PROGRAM F01_METS_SingleInputs
VAR
(*METS General Filtered Inputs FB ***************************************************************************************************************)

	fbMestStart				: 	FB_IO2_SingleInputCtrl;
	fbMestStop				: 	FB_IO2_SingleInputCtrl;
	fbMestReset				:	FB_IO2_SingleInputCtrl;

	fbMETS_24VPowerSupplyOK		: FB_IO2_SingleInputCtrl;
	fbTPD24VPowerSupplyOK			: FB_IO2_SingleInputCtrl;
	fbAirPressureOK				: FB_IO2_SingleInputCtrl;
	fbAirConditionerOK				: FB_IO2_SingleInputCtrl; (**)
	fbUPSBatteryAlarm				: FB_IO2_SingleInputCtrl;
	fbNetworkOKFromSwitch			: FB_IO2_SingleInputCtrl;


	fbPreMachineAutoRun			: FB_IO2_SingleInputCtrl;
	fbCasePackerAutoRun			: FB_IO2_SingleInputCtrl;

	fbDoorOpenZone1				: FB_IO2_SingleInputCtrl;
	fbDoorOpenZone2 				: FB_IO2_SingleInputCtrl;

	fbAuxRowCompleteSesnor			: FB_IO2_SingleInputCtrl;
	fbCaseAtRejectStation	 		: FB_IO2_SingleInputCtrl;
	fbCaseRejectedByCasePacker		: FB_IO2_SingleInputCtrl;
	fbCaseContentValidationComplete	: FB_IO2_SingleInputCtrl;
	fbCaseLeavingPrintArea			: FB_IO2_SingleInputCtrl;

(*METS CX UPS  Filtered Inputs  FB***************************************************************************************************************)
	fbMainSupplyHealthy			:	FB_IO2_SingleInputCtrl;	(*ib64KF1_1_MainsSupplyHealthy*)
	fbUPSHealthy					:	FB_IO2_SingleInputCtrl;	(*ib64KF1_5_UPSHealthy*)
	fbUPSBatteryMode				:	FB_IO2_SingleInputCtrl;	(*ib64KF1_2_UPSBatteryMode*)
	fbUPSBatteryCharging			:	FB_IO2_SingleInputCtrl;	(*ib64KF1_6_UPSBatteryCharging*)


(*METS Camera Filtered Inputs  FB***************************************************************************************************************)

	fbCamera01TrigSensor			: FB_IO2_SingleInputCtrl;
	fbCamera02TrigSensor			: FB_IO2_SingleInputCtrl;
	fbCamera03TrigSensor			: FB_IO2_SingleInputCtrl;
	fbCamera04TrigSensor			: FB_IO2_SingleInputCtrl;
	fbCamera05TrigSensor			: FB_IO2_SingleInputCtrl;
	fbCamera06TrigSensor			: FB_IO2_SingleInputCtrl;
	fbCamera07TrigSensor			: FB_IO2_SingleInputCtrl;
	fbCamera08TrigSensor			: FB_IO2_SingleInputCtrl;
	fbCamera09TrigSensor			: FB_IO2_SingleInputCtrl;
	fbCamera10TrigSensor			: FB_IO2_SingleInputCtrl;
	fbCamera11TrigSensor			: FB_IO2_SingleInputCtrl;
	fbCamera12TrigSensor			: FB_IO2_SingleInputCtrl;

(*METS Casepacker  Filtered Inputs  FB***************************************************************************************************************)

	fbEUCABuildBackPreMachine		: FB_IO2_SingleInputCtrl;
	fbEUCAExitBlocked				: FB_IO2_SingleInputCtrl; (**)

	fbOuterAtSystemInfeed		: FB_IO2_SingleInputCtrl;
	fbOuterAtAdditionalConv		: FB_IO2_SingleInputCtrl;

	fbQAButtonReject				: FB_IO2_SingleInputCtrl;
	fbOuterAtRejectStation 			: FB_IO2_SingleInputCtrl;
	fbOuterRejectConfirm			: FB_IO2_SingleInputCtrl;
	fbRejectBinFull					: FB_IO2_SingleInputCtrl;


	(*Transfer Conveyor*)
	fbTransferCoveyorDoorGuard1		: FB_IO2_SingleInputCtrl;
	fbTransferCoveyorDoorGuard2		: FB_IO2_SingleInputCtrl;

	fbTransferConveyorPlugConnected	: FB_IO2_SingleInputCtrl;
	fbOutfeedConveyorPlugConnected	: FB_IO2_SingleInputCtrl;
	fbAdditionalConveyorPlugConnected	: FB_IO2_SingleInputCtrl;



(*METS Cylinders Filtered Inputs  FB***************************************************************************************************************)

	fbClampCylinderExtended		: FB_IO2_SingleInputCtrl;
	fbClampCylinderRetracted		: FB_IO2_SingleInputCtrl;

	fbGateCylinderExtended			: FB_IO2_SingleInputCtrl;
	fbGateCylinderRetracted 			: FB_IO2_SingleInputCtrl;

	fbRejectCylinderExtended		: FB_IO2_SingleInputCtrl;
	fbRejectCylinderRetracted 		: FB_IO2_SingleInputCtrl;

	fbAdditionalRejectCylinderExtended		: FB_IO2_SingleInputCtrl;
	fbAdditionalRejectCylinderRetracted 		: FB_IO2_SingleInputCtrl;

	fbFirstPusherCylinderExtended		: FB_IO2_SingleInputCtrl;
	fbFirstPusherCylinderRetracted 		: FB_IO2_SingleInputCtrl;

	fbSecondPusherCylinderExtended		: FB_IO2_SingleInputCtrl;
	fbSecondPusherCylinderRetracted 		: FB_IO2_SingleInputCtrl;

(*METS SFLX Machine Filtered Inputs  FB***************************************************************************************************************)

	fbOuterInfeedJam						: FB_IO2_SingleInputCtrl;
	fbOuterTransferConfirmation			: FB_IO2_SingleInputCtrl;
	fbRejectConfirmationNCW				: FB_IO2_SingleInputCtrl;
	fbRejectBinFullNCW					: FB_IO2_SingleInputCtrl;
	fbOuterAtTransferReject				: FB_IO2_SingleInputCtrl;
	fbOuterAtSideFlexExit					: FB_IO2_SingleInputCtrl;
	fbOuterAtPostMachineInfeed			: FB_IO2_SingleInputCtrl;

	fbGuard1FlexInfeedDoor	  	: FB_IO2_SingleInputCtrl;
	fbGuard3FlexRHDoor		: FB_IO2_SingleInputCtrl;
	fbGuard4FlexPrinterDoor		: FB_IO2_SingleInputCtrl;
	fbGuard5FlexLHDoor		: FB_IO2_SingleInputCtrl;

(*METS CML Filtered Inputs ***************************************************************************************************************)

	fbGuard1UpperSideAccessDoor	: FB_IO2_SingleInputCtrl;
	fbGuard2UpperDoorLabellerSide	: FB_IO2_SingleInputCtrl;
	fbGuard3OutfeedTunnel			: FB_IO2_SingleInputCtrl;
	fbGuard4ElectricalBoxInPosition	: FB_IO2_SingleInputCtrl;
	fbGuard5RejectBinLHSide			: FB_IO2_SingleInputCtrl;
	fbGuard6RejectBinRHSide			: FB_IO2_SingleInputCtrl;
	fbGuard7HTTDoorGuard			: FB_IO2_SingleInputCtrl;
	fbGuard10FrontUpperDoor			: FB_IO2_SingleInputCtrl;
	fbGuard11GuardLowerLabellerSide	: FB_IO2_SingleInputCtrl;

	fbRejectBinGuardIsReset			: FB_IO2_SingleInputCtrl;
	fbLabeller1GuardIsReset			: FB_IO2_SingleInputCtrl;
	fbLabeller2GuardIsReset			: FB_IO2_SingleInputCtrl;

	fbResetPB							: FB_IO2_SingleInputCtrl;

	fbOuterAtCMLRejectStation		: FB_IO2_SingleInputLockCtrl;

	fbRotaryTransferPackAtStopPlate		: FB_IO2_SingleInputCtrl;
	fbRotaryTransferTorqueLimiter		: FB_IO2_SingleInputCtrl;
	fbRotaryTransferDelayStop1			: FB_IO2_SingleInputCtrl;
	fbRotaryTransferDelayStop2			: FB_IO2_SingleInputCtrl;

	fbLoweratorGuideRHLowerInPosition	: FB_IO2_SingleInputCtrl;
	fbLoweratorGuideLHLowerInPosition	: FB_IO2_SingleInputCtrl;

	fbAdditionalConveyor1Isolator		: FB_IO2_SingleInputCtrl;
	fbAdditionalConveyor2Isolator		: FB_IO2_SingleInputCtrl;
	fbAdditionalConveyor3Isolator		: FB_IO2_SingleInputCtrl;
	fbAdditionalConveyor4Isolator		: FB_IO2_SingleInputCtrl;

	fbAdditionalConveyor4OK				: FB_IO2_SingleInputCtrl;

	fbConveyorIndexContact				: FB_IO2_SingleInputCtrl;

(*METS SADDLE (Gating&Reject System) Filtered Inputs  FB***************************************************************************************************************)

	fbOuterAtClamp						: FB_IO2_SingleInputCtrl;
	fbOuterAtLabelGate						: FB_IO2_SingleInputCtrl;

	fbSaddlePressureOK					: FB_IO2_SingleInputCtrl;

	fbGateImpactSensor					: FB_IO2_SingleInputCtrl;
	fbGateClear							 : FB_IO2_SingleInputCtrl;

(*METS PLAS/NCW Machine Filtered Inputs  FB***************************************************************************************************************)
	(*Wrapper*)
	fbMasterlistDoorGuard1					: FB_IO2_SingleInputCtrl;
	fbMasterlistDoorGuard2					: FB_IO2_SingleInputCtrl;
	fbMasterlistDoorGuard3					: FB_IO2_SingleInputCtrl;

	fbOuterBrushOpen							: FB_IO2_SingleInputCtrl;
	fbPackAggregationDoorGuard1			: FB_IO2_SingleInputCtrl;
	fbPackAggregationDoorGuard2			: FB_IO2_SingleInputCtrl;

	fbWrapperDoorGuard1						: FB_IO2_SingleInputCtrl;
	fbWrapperDoorGuard2						: FB_IO2_SingleInputCtrl;

	fbHeatTunelPackReject					: FB_IO2_SingleInputCtrl;
	fbWrapperPackReject						: FB_IO2_SingleInputCtrl;
	fbWrapperPackReject2						: FB_IO2_SingleInputCtrl;
	fbWrapperOuterComplete					: FB_IO2_SingleInputCtrl;

	fbFilmInPosition 							: FB_IO2_SingleInputCtrl;
	fbInhibitIntermediateCamera 				: FB_IO2_SingleInputCtrl;
	fbIntermediatePrinterTrigger				: FB_IO2_SingleInputCtrl;

(*METS Labeller Filtered Inputs ***************************************************************************************************************)

	fbLabeller1InPosition					: FB_IO2_SingleInputCtrl;
	fbLabeller1OuterAtLabeller			: FB_IO2_SingleInputLockCtrl;(*: FB_IO2_SingleInputCtrl;*)

	fbLabeller1Ready						: FB_IO2_SingleInputCtrl;
	fbLabeller1DataReady					: FB_IO2_SingleInputCtrl;
	fbLabeller1HomePosition				: FB_IO2_SingleInputCtrl;
	fbLabeller1LabelPrinted				: FB_IO2_SingleInputCtrl;
	fbLabeller1ReadyToApply				: FB_IO2_SingleInputCtrl;
	fbLabeller1ApplyDone					: FB_IO2_SingleInputCtrl;
	fbLabeller1SummaryWarning			: FB_IO2_SingleInputCtrl;
	fbLabeller1Error						: FB_IO2_SingleInputCtrl;

	fbLabeller2InPosition					: FB_IO2_SingleInputCtrl;
	fbLabeller2OuterAtLabeller			: FB_IO2_SingleInputLockCtrl;(*: FB_IO2_SingleInputCtrl;*)

	fbLabeller2Ready						: FB_IO2_SingleInputCtrl;
	fbLabeller2DataReady					: FB_IO2_SingleInputCtrl;
	fbLabeller2HomePosition				: FB_IO2_SingleInputCtrl;
	fbLabeller2LabelPrinted				: FB_IO2_SingleInputCtrl;
	fbLabeller2ReadyToApply				: FB_IO2_SingleInputCtrl;
	fbLabeller2ApplyDone					: FB_IO2_SingleInputCtrl;
	fbLabeller2SummaryWarning			: FB_IO2_SingleInputCtrl;
	fbLabeller2Error						: FB_IO2_SingleInputCtrl;

(*METS PAOL  Filtered Inputs  FB***************************************************************************************************************)

	fbPreMachineBuildBack			: FB_IO2_SingleInputCtrl;
	fbTPDExitBlocked				: FB_IO2_SingleInputCtrl;
(*	fbInfeedConveyorStart			: FB_IO2_SingleInputCtrl;*)
	fbPackSeparationDriveOK			: FB_IO2_SingleInputCtrl;
	fbInfeedConveyorDriveOK		: FB_IO2_SingleInputCtrl;

	fbPackAggregCameraRigSensor		: FB_IO2_SingleInputCtrl;
	fbPackIsolatorDrive				: FB_IO2_SingleInputCtrl;


(**********************************************************************************************************************************)

	fbDebugCNT							: FB_DEBUG_CounterArray;
	aCNTDebug							: ARRAY [1..10] OF UDINT;
	bResetCNT							: BOOL;

	bTestConvRun	: BOOL;



END_VAR

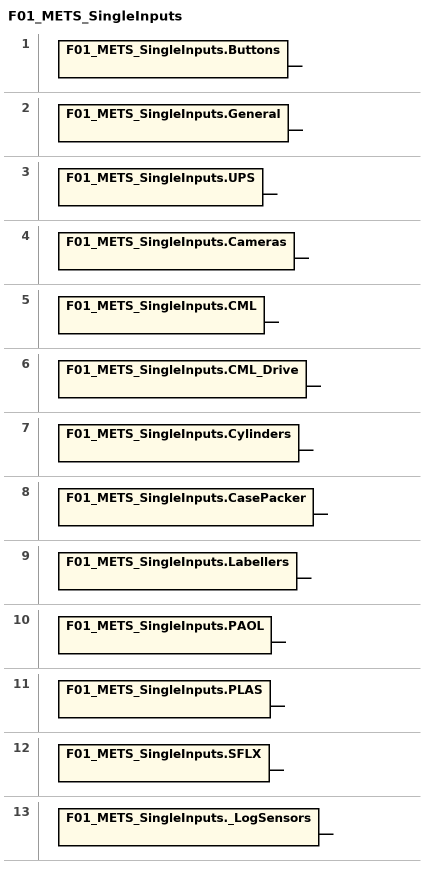
// NETWORK 1
F01_METS_SingleInputs.Buttons();

// NETWORK 2
F01_METS_SingleInputs.General();

// NETWORK 3
F01_METS_SingleInputs.UPS();

// NETWORK 4
F01_METS_SingleInputs.Cameras();

// NETWORK 5
F01_METS_SingleInputs.CML();

// NETWORK 6
F01_METS_SingleInputs.CML_Drive();

// NETWORK 7
F01_METS_SingleInputs.Cylinders();

// NETWORK 8
F01_METS_SingleInputs.CasePacker();

// NETWORK 9
F01_METS_SingleInputs.Labellers();

// NETWORK 10
F01_METS_SingleInputs.PAOL();

// NETWORK 11
F01_METS_SingleInputs.PLAS();

// NETWORK 12
F01_METS_SingleInputs.SFLX();

// NETWORK 13
F01_METS_SingleInputs._LogSensors();

ACTION _LogSensors:
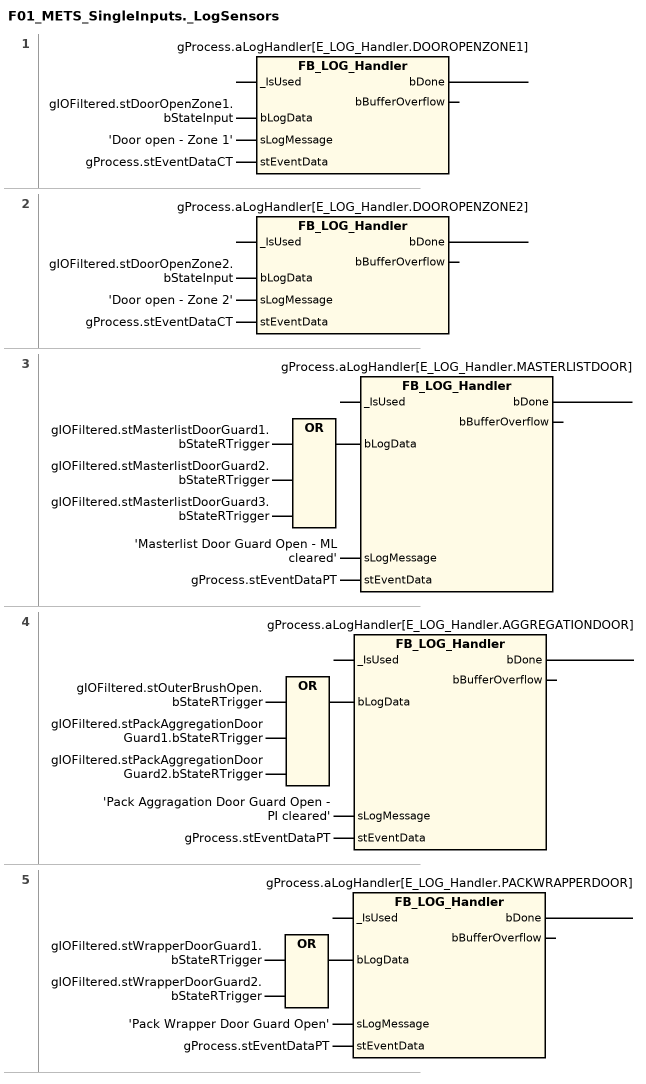
// NETWORK 1
gProcess.aLogHandler[E_LOG_Handler.DOOROPENZONE1](
    bLogData := gIOFiltered.stDoorOpenZone1.bStateInput,
    sLogMessage := 'Door open - Zone 1',
    stEventData := gProcess.stEventDataCT); // FB_LOG_Handler

// NETWORK 2
gProcess.aLogHandler[E_LOG_Handler.DOOROPENZONE2](
    bLogData := gIOFiltered.stDoorOpenZone2.bStateInput,
    sLogMessage := 'Door open - Zone 2',
    stEventData := gProcess.stEventDataCT); // FB_LOG_Handler

// NETWORK 3
gProcess.aLogHandler[E_LOG_Handler.MASTERLISTDOOR](
    bLogData := gIOFiltered.stMasterlistDoorGuard1.bStateRTrigger OR gIOFiltered.stMasterlistDoorGuard2.bStateRTrigger OR gIOFiltered.stMasterlistDoorGuard3.bStateRTrigger,
    sLogMessage := 'Masterlist Door Guard Open - ML cleared',
    stEventData := gProcess.stEventDataPT); // FB_LOG_Handler

// NETWORK 4
gProcess.aLogHandler[E_LOG_Handler.AGGREGATIONDOOR](
    bLogData := gIOFiltered.stOuterBrushOpen.bStateRTrigger OR gIOFiltered.stPackAggregationDoorGuard1.bStateRTrigger OR gIOFiltered.stPackAggregationDoorGuard2.bStateRTrigger,
    sLogMessage := 'Pack Aggragation Door Guard Open - PI cleared',
    stEventData := gProcess.stEventDataPT); // FB_LOG_Handler

// NETWORK 5
gProcess.aLogHandler[E_LOG_Handler.PACKWRAPPERDOOR](
    bLogData := gIOFiltered.stWrapperDoorGuard1.bStateRTrigger OR gIOFiltered.stWrapperDoorGuard2.bStateRTrigger,
    sLogMessage := 'Pack Wrapper Door Guard Open',
    stEventData := gProcess.stEventDataPT); // FB_LOG_Handler
END_ACTION

ACTION Buttons:
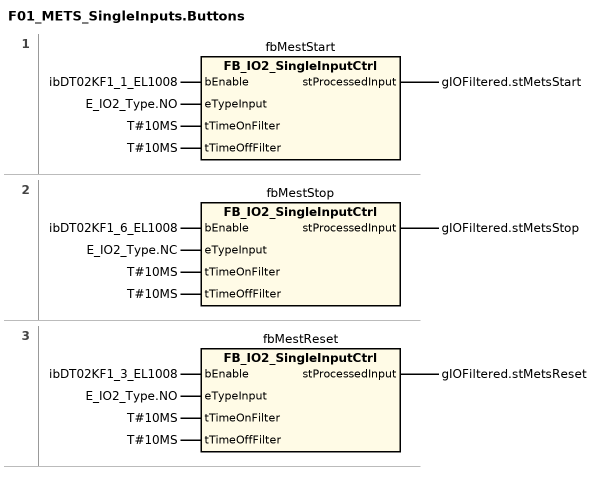
// NETWORK 1
fbMestStart(
    bEnable := ibDT02KF1_1_EL1008,
    eTypeInput := E_IO2_Type.NO,
    tTimeOnFilter := T#10MS,
    tTimeOffFilter := T#10MS); // FB_IO2_SingleInputCtrl
gIOFiltered.stMetsStart := fbMestStart.stProcessedInput;

// NETWORK 2
fbMestStop(
    bEnable := ibDT02KF1_6_EL1008,
    eTypeInput := E_IO2_Type.NC,
    tTimeOnFilter := T#10MS,
    tTimeOffFilter := T#10MS); // FB_IO2_SingleInputCtrl
gIOFiltered.stMetsStop := fbMestStop.stProcessedInput;

// NETWORK 3
fbMestReset(
    bEnable := ibDT02KF1_3_EL1008,
    eTypeInput := E_IO2_Type.NO,
    tTimeOnFilter := T#10MS,
    tTimeOffFilter := T#10MS); // FB_IO2_SingleInputCtrl
gIOFiltered.stMetsReset := fbMestReset.stProcessedInput;
END_ACTION

ACTION Cameras:
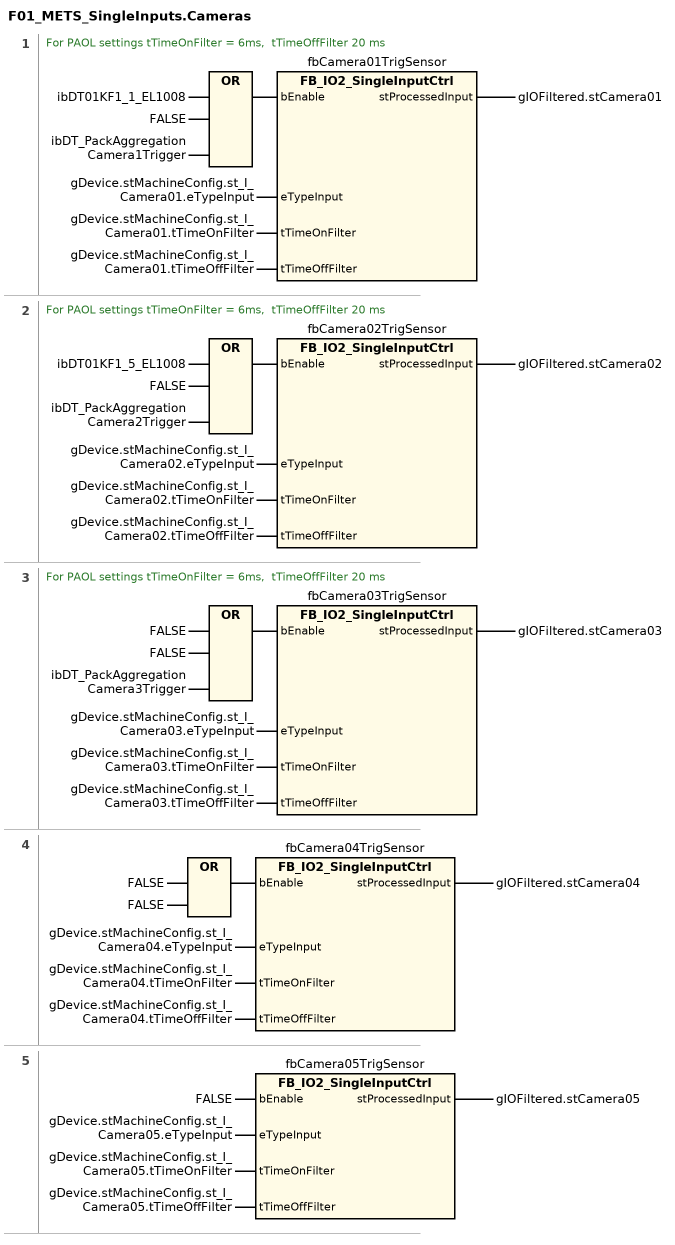
// NETWORK 1
// For PAOL settings tTimeOnFilter = 6ms,  tTimeOffFilter 20 ms
fbCamera01TrigSensor(
    bEnable := ibDT01KF1_1_EL1008 OR FALSE OR ibDT_PackAggregationCamera1Trigger,
    eTypeInput := gDevice.stMachineConfig.st_I_Camera01.eTypeInput,
    tTimeOnFilter := gDevice.stMachineConfig.st_I_Camera01.tTimeOnFilter,
    tTimeOffFilter := gDevice.stMachineConfig.st_I_Camera01.tTimeOffFilter); // FB_IO2_SingleInputCtrl
gIOFiltered.stCamera01 := fbCamera01TrigSensor.stProcessedInput;

// NETWORK 2
// For PAOL settings tTimeOnFilter = 6ms,  tTimeOffFilter 20 ms
fbCamera02TrigSensor(
    bEnable := ibDT01KF1_5_EL1008 OR FALSE OR ibDT_PackAggregationCamera2Trigger,
    eTypeInput := gDevice.stMachineConfig.st_I_Camera02.eTypeInput,
    tTimeOnFilter := gDevice.stMachineConfig.st_I_Camera02.tTimeOnFilter,
    tTimeOffFilter := gDevice.stMachineConfig.st_I_Camera02.tTimeOffFilter); // FB_IO2_SingleInputCtrl
gIOFiltered.stCamera02 := fbCamera02TrigSensor.stProcessedInput;

// NETWORK 3
// For PAOL settings tTimeOnFilter = 6ms,  tTimeOffFilter 20 ms
fbCamera03TrigSensor(
    bEnable := FALSE OR FALSE OR ibDT_PackAggregationCamera3Trigger,
    eTypeInput := gDevice.stMachineConfig.st_I_Camera03.eTypeInput,
    tTimeOnFilter := gDevice.stMachineConfig.st_I_Camera03.tTimeOnFilter,
    tTimeOffFilter := gDevice.stMachineConfig.st_I_Camera03.tTimeOffFilter); // FB_IO2_SingleInputCtrl
gIOFiltered.stCamera03 := fbCamera03TrigSensor.stProcessedInput;

// NETWORK 4
fbCamera04TrigSensor(
    bEnable := FALSE OR FALSE,
    eTypeInput := gDevice.stMachineConfig.st_I_Camera04.eTypeInput,
    tTimeOnFilter := gDevice.stMachineConfig.st_I_Camera04.tTimeOnFilter,
    tTimeOffFilter := gDevice.stMachineConfig.st_I_Camera04.tTimeOffFilter); // FB_IO2_SingleInputCtrl
gIOFiltered.stCamera04 := fbCamera04TrigSensor.stProcessedInput;

// NETWORK 5
fbCamera05TrigSensor(
    bEnable := FALSE,
    eTypeInput := gDevice.stMachineConfig.st_I_Camera05.eTypeInput,
    tTimeOnFilter := gDevice.stMachineConfig.st_I_Camera05.tTimeOnFilter,
    tTimeOffFilter := gDevice.stMachineConfig.st_I_Camera05.tTimeOffFilter); // FB_IO2_SingleInputCtrl
gIOFiltered.stCamera05 := fbCamera05TrigSensor.stProcessedInput;

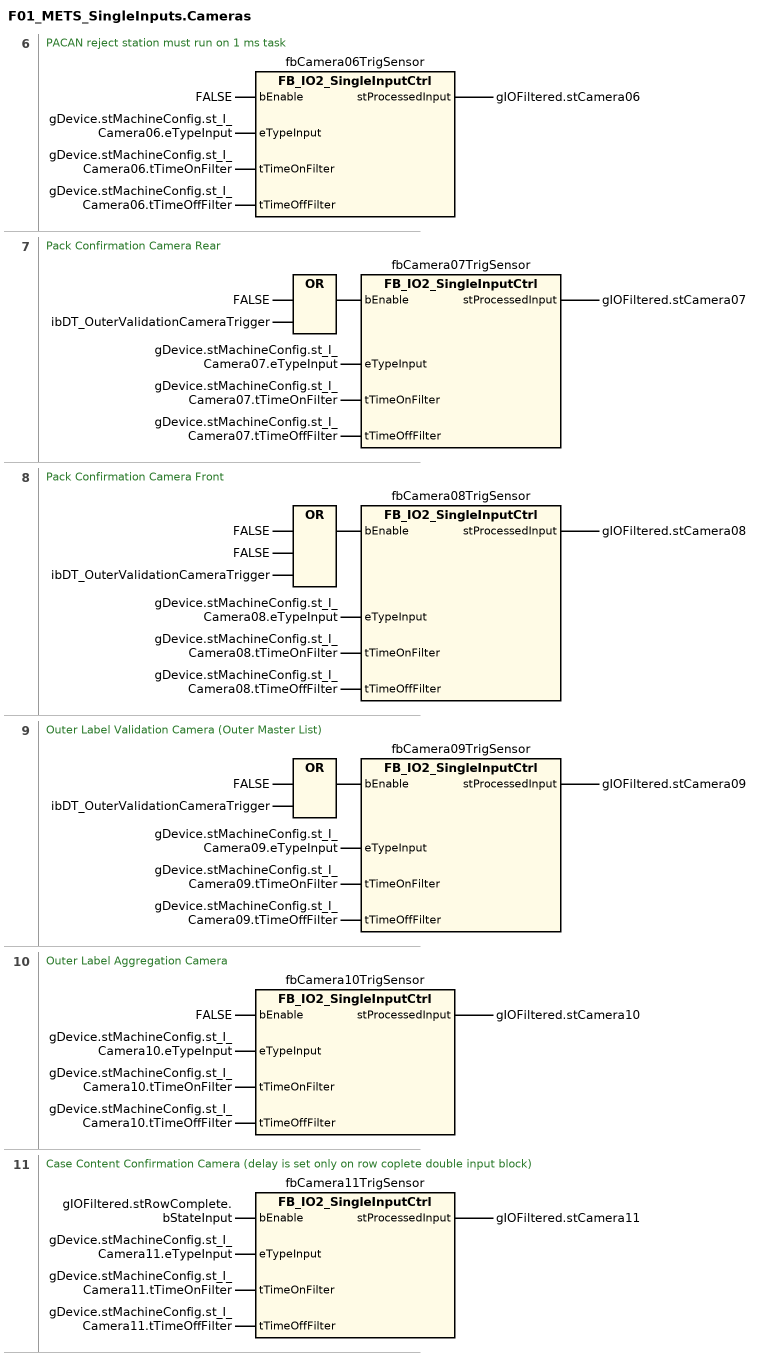
// NETWORK 6
// PACAN reject station must run on 1 ms task
fbCamera06TrigSensor(
    bEnable := FALSE,
    eTypeInput := gDevice.stMachineConfig.st_I_Camera06.eTypeInput,
    tTimeOnFilter := gDevice.stMachineConfig.st_I_Camera06.tTimeOnFilter,
    tTimeOffFilter := gDevice.stMachineConfig.st_I_Camera06.tTimeOffFilter); // FB_IO2_SingleInputCtrl
gIOFiltered.stCamera06 := fbCamera06TrigSensor.stProcessedInput;

// NETWORK 7
// Pack Confirmation Camera Rear
fbCamera07TrigSensor(
    bEnable := FALSE OR ibDT_OuterValidationCameraTrigger,
    eTypeInput := gDevice.stMachineConfig.st_I_Camera07.eTypeInput,
    tTimeOnFilter := gDevice.stMachineConfig.st_I_Camera07.tTimeOnFilter,
    tTimeOffFilter := gDevice.stMachineConfig.st_I_Camera07.tTimeOffFilter); // FB_IO2_SingleInputCtrl
gIOFiltered.stCamera07 := fbCamera07TrigSensor.stProcessedInput;

// NETWORK 8
// Pack Confirmation Camera Front
fbCamera08TrigSensor(
    bEnable := FALSE OR FALSE OR ibDT_OuterValidationCameraTrigger,
    eTypeInput := gDevice.stMachineConfig.st_I_Camera08.eTypeInput,
    tTimeOnFilter := gDevice.stMachineConfig.st_I_Camera08.tTimeOnFilter,
    tTimeOffFilter := gDevice.stMachineConfig.st_I_Camera08.tTimeOffFilter); // FB_IO2_SingleInputCtrl
gIOFiltered.stCamera08 := fbCamera08TrigSensor.stProcessedInput;

// NETWORK 9
// Outer Label Validation Camera (Outer Master List)
fbCamera09TrigSensor(
    bEnable := FALSE OR ibDT_OuterValidationCameraTrigger,
    eTypeInput := gDevice.stMachineConfig.st_I_Camera09.eTypeInput,
    tTimeOnFilter := gDevice.stMachineConfig.st_I_Camera09.tTimeOnFilter,
    tTimeOffFilter := gDevice.stMachineConfig.st_I_Camera09.tTimeOffFilter); // FB_IO2_SingleInputCtrl
gIOFiltered.stCamera09 := fbCamera09TrigSensor.stProcessedInput;

// NETWORK 10
// Outer Label Aggregation Camera
fbCamera10TrigSensor(
    bEnable := FALSE,
    eTypeInput := gDevice.stMachineConfig.st_I_Camera10.eTypeInput,
    tTimeOnFilter := gDevice.stMachineConfig.st_I_Camera10.tTimeOnFilter,
    tTimeOffFilter := gDevice.stMachineConfig.st_I_Camera10.tTimeOffFilter); // FB_IO2_SingleInputCtrl
gIOFiltered.stCamera10 := fbCamera10TrigSensor.stProcessedInput;

// NETWORK 11
// Case Content Confirmation Camera (delay is set only on row coplete double input block)
fbCamera11TrigSensor(
    bEnable := gIOFiltered.stRowComplete.bStateInput,
    eTypeInput := gDevice.stMachineConfig.st_I_Camera11.eTypeInput,
    tTimeOnFilter := gDevice.stMachineConfig.st_I_Camera11.tTimeOnFilter,
    tTimeOffFilter := gDevice.stMachineConfig.st_I_Camera11.tTimeOffFilter); // FB_IO2_SingleInputCtrl
gIOFiltered.stCamera11 := fbCamera11TrigSensor.stProcessedInput;

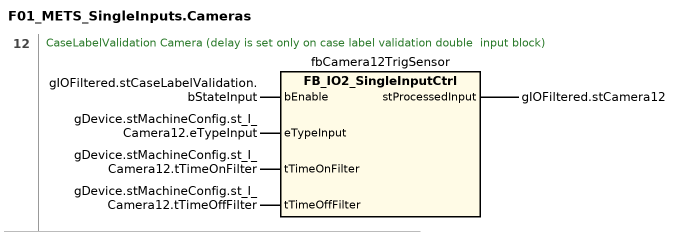
// NETWORK 12
// CaseLabelValidation Camera (delay is set only on case label validation double  input block)
fbCamera12TrigSensor(
    bEnable := gIOFiltered.stCaseLabelValidation.bStateInput,
    eTypeInput := gDevice.stMachineConfig.st_I_Camera12.eTypeInput,
    tTimeOnFilter := gDevice.stMachineConfig.st_I_Camera12.tTimeOnFilter,
    tTimeOffFilter := gDevice.stMachineConfig.st_I_Camera12.tTimeOffFilter); // FB_IO2_SingleInputCtrl
gIOFiltered.stCamera12 := fbCamera12TrigSensor.stProcessedInput;
END_ACTION

ACTION CasePacker:
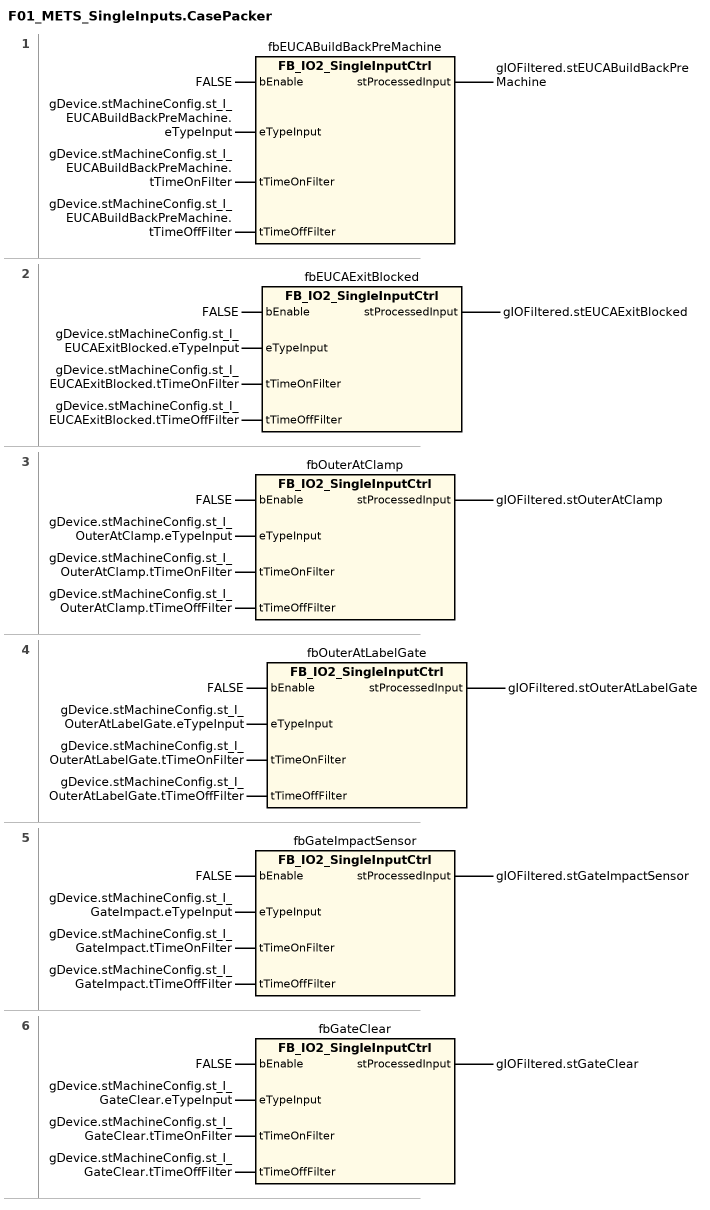
// NETWORK 1
fbEUCABuildBackPreMachine(
    bEnable := FALSE,
    eTypeInput := gDevice.stMachineConfig.st_I_EUCABuildBackPreMachine.eTypeInput,
    tTimeOnFilter := gDevice.stMachineConfig.st_I_EUCABuildBackPreMachine.tTimeOnFilter,
    tTimeOffFilter := gDevice.stMachineConfig.st_I_EUCABuildBackPreMachine.tTimeOffFilter); // FB_IO2_SingleInputCtrl
gIOFiltered.stEUCABuildBackPreMachine := fbEUCABuildBackPreMachine.stProcessedInput;

// NETWORK 2
fbEUCAExitBlocked(
    bEnable := FALSE,
    eTypeInput := gDevice.stMachineConfig.st_I_EUCAExitBlocked.eTypeInput,
    tTimeOnFilter := gDevice.stMachineConfig.st_I_EUCAExitBlocked.tTimeOnFilter,
    tTimeOffFilter := gDevice.stMachineConfig.st_I_EUCAExitBlocked.tTimeOffFilter); // FB_IO2_SingleInputCtrl
gIOFiltered.stEUCAExitBlocked := fbEUCAExitBlocked.stProcessedInput;

// NETWORK 3
fbOuterAtClamp(
    bEnable := FALSE,
    eTypeInput := gDevice.stMachineConfig.st_I_OuterAtClamp.eTypeInput,
    tTimeOnFilter := gDevice.stMachineConfig.st_I_OuterAtClamp.tTimeOnFilter,
    tTimeOffFilter := gDevice.stMachineConfig.st_I_OuterAtClamp.tTimeOffFilter); // FB_IO2_SingleInputCtrl
gIOFiltered.stOuterAtClamp := fbOuterAtClamp.stProcessedInput;

// NETWORK 4
fbOuterAtLabelGate(
    bEnable := FALSE,
    eTypeInput := gDevice.stMachineConfig.st_I_OuterAtLabelGate.eTypeInput,
    tTimeOnFilter := gDevice.stMachineConfig.st_I_OuterAtLabelGate.tTimeOnFilter,
    tTimeOffFilter := gDevice.stMachineConfig.st_I_OuterAtLabelGate.tTimeOffFilter); // FB_IO2_SingleInputCtrl
gIOFiltered.stOuterAtLabelGate := fbOuterAtLabelGate.stProcessedInput;

// NETWORK 5
fbGateImpactSensor(
    bEnable := FALSE,
    eTypeInput := gDevice.stMachineConfig.st_I_GateImpact.eTypeInput,
    tTimeOnFilter := gDevice.stMachineConfig.st_I_GateImpact.tTimeOnFilter,
    tTimeOffFilter := gDevice.stMachineConfig.st_I_GateImpact.tTimeOffFilter); // FB_IO2_SingleInputCtrl
gIOFiltered.stGateImpactSensor := fbGateImpactSensor.stProcessedInput;

// NETWORK 6
fbGateClear(
    bEnable := FALSE,
    eTypeInput := gDevice.stMachineConfig.st_I_GateClear.eTypeInput,
    tTimeOnFilter := gDevice.stMachineConfig.st_I_GateClear.tTimeOnFilter,
    tTimeOffFilter := gDevice.stMachineConfig.st_I_GateClear.tTimeOffFilter); // FB_IO2_SingleInputCtrl
gIOFiltered.stGateClear := fbGateClear.stProcessedInput;

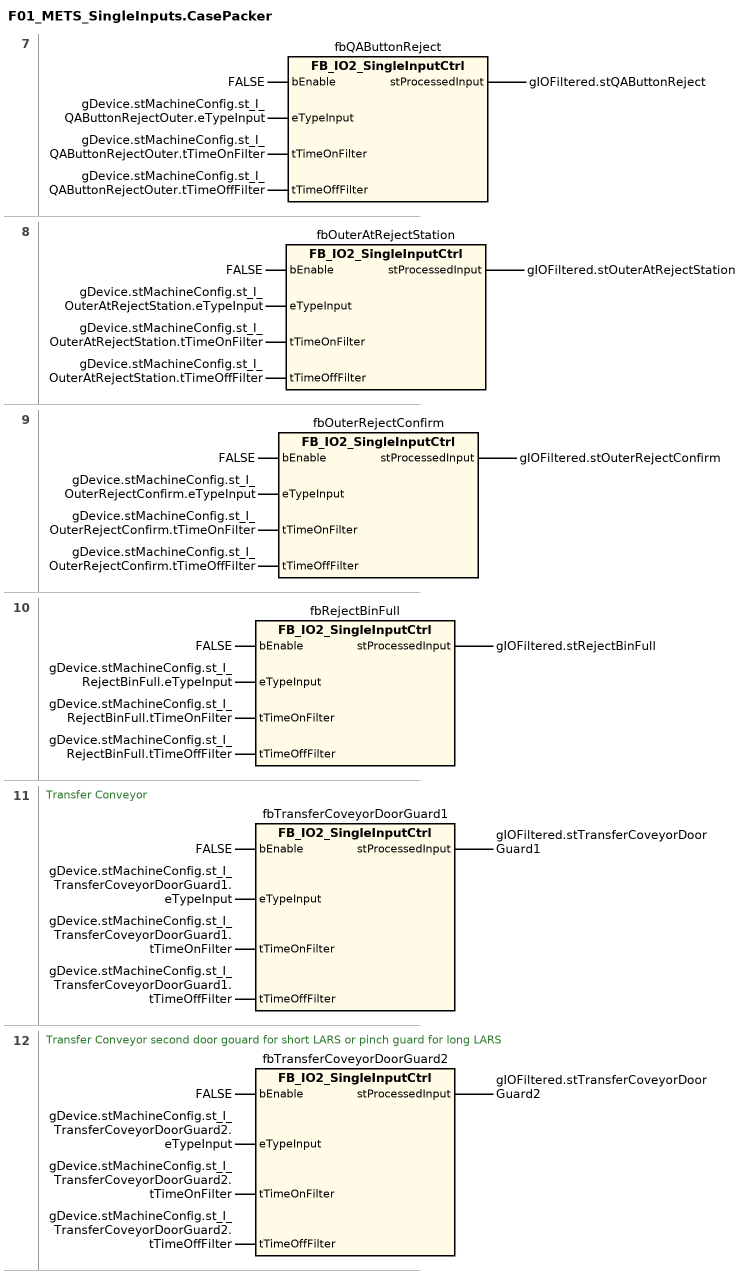
// NETWORK 7
fbQAButtonReject(
    bEnable := FALSE,
    eTypeInput := gDevice.stMachineConfig.st_I_QAButtonRejectOuter.eTypeInput,
    tTimeOnFilter := gDevice.stMachineConfig.st_I_QAButtonRejectOuter.tTimeOnFilter,
    tTimeOffFilter := gDevice.stMachineConfig.st_I_QAButtonRejectOuter.tTimeOffFilter); // FB_IO2_SingleInputCtrl
gIOFiltered.stQAButtonReject := fbQAButtonReject.stProcessedInput;

// NETWORK 8
fbOuterAtRejectStation(
    bEnable := FALSE,
    eTypeInput := gDevice.stMachineConfig.st_I_OuterAtRejectStation.eTypeInput,
    tTimeOnFilter := gDevice.stMachineConfig.st_I_OuterAtRejectStation.tTimeOnFilter,
    tTimeOffFilter := gDevice.stMachineConfig.st_I_OuterAtRejectStation.tTimeOffFilter); // FB_IO2_SingleInputCtrl
gIOFiltered.stOuterAtRejectStation := fbOuterAtRejectStation.stProcessedInput;

// NETWORK 9
fbOuterRejectConfirm(
    bEnable := FALSE,
    eTypeInput := gDevice.stMachineConfig.st_I_OuterRejectConfirm.eTypeInput,
    tTimeOnFilter := gDevice.stMachineConfig.st_I_OuterRejectConfirm.tTimeOnFilter,
    tTimeOffFilter := gDevice.stMachineConfig.st_I_OuterRejectConfirm.tTimeOffFilter); // FB_IO2_SingleInputCtrl
gIOFiltered.stOuterRejectConfirm := fbOuterRejectConfirm.stProcessedInput;

// NETWORK 10
fbRejectBinFull(
    bEnable := FALSE,
    eTypeInput := gDevice.stMachineConfig.st_I_RejectBinFull.eTypeInput,
    tTimeOnFilter := gDevice.stMachineConfig.st_I_RejectBinFull.tTimeOnFilter,
    tTimeOffFilter := gDevice.stMachineConfig.st_I_RejectBinFull.tTimeOffFilter); // FB_IO2_SingleInputCtrl
gIOFiltered.stRejectBinFull := fbRejectBinFull.stProcessedInput;

// NETWORK 11
// Transfer Conveyor
fbTransferCoveyorDoorGuard1(
    bEnable := FALSE,
    eTypeInput := gDevice.stMachineConfig.st_I_TransferCoveyorDoorGuard1.eTypeInput,
    tTimeOnFilter := gDevice.stMachineConfig.st_I_TransferCoveyorDoorGuard1.tTimeOnFilter,
    tTimeOffFilter := gDevice.stMachineConfig.st_I_TransferCoveyorDoorGuard1.tTimeOffFilter); // FB_IO2_SingleInputCtrl
gIOFiltered.stTransferCoveyorDoorGuard1 := fbTransferCoveyorDoorGuard1.stProcessedInput;

// NETWORK 12
// Transfer Conveyor second door gouard for short LARS or pinch guard for long LARS
fbTransferCoveyorDoorGuard2(
    bEnable := FALSE,
    eTypeInput := gDevice.stMachineConfig.st_I_TransferCoveyorDoorGuard2.eTypeInput,
    tTimeOnFilter := gDevice.stMachineConfig.st_I_TransferCoveyorDoorGuard2.tTimeOnFilter,
    tTimeOffFilter := gDevice.stMachineConfig.st_I_TransferCoveyorDoorGuard2.tTimeOffFilter); // FB_IO2_SingleInputCtrl
gIOFiltered.stTransferCoveyorDoorGuard2 := fbTransferCoveyorDoorGuard2.stProcessedInput;

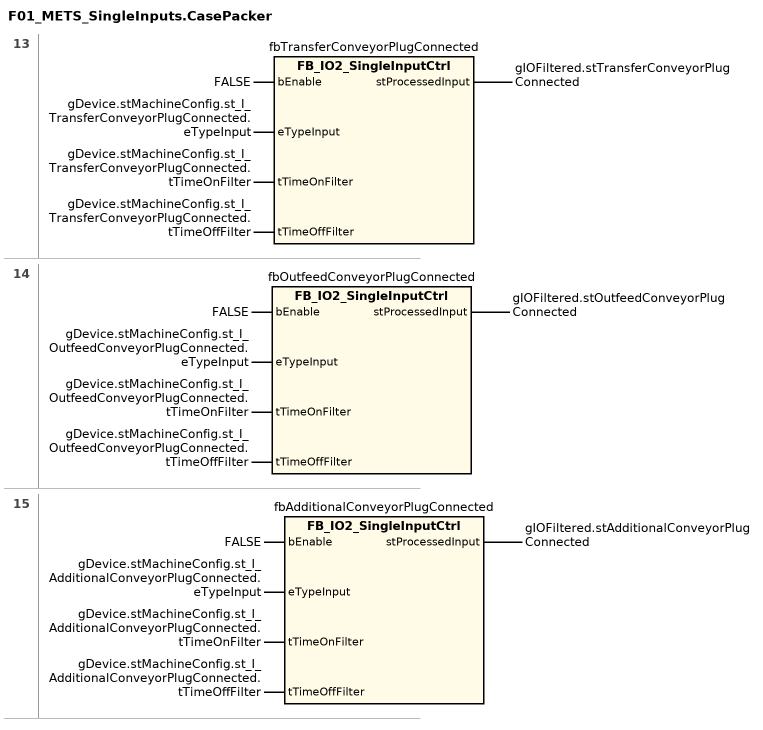
// NETWORK 13
fbTransferConveyorPlugConnected(
    bEnable := FALSE,
    eTypeInput := gDevice.stMachineConfig.st_I_TransferConveyorPlugConnected.eTypeInput,
    tTimeOnFilter := gDevice.stMachineConfig.st_I_TransferConveyorPlugConnected.tTimeOnFilter,
    tTimeOffFilter := gDevice.stMachineConfig.st_I_TransferConveyorPlugConnected.tTimeOffFilter); // FB_IO2_SingleInputCtrl
gIOFiltered.stTransferConveyorPlugConnected := fbTransferConveyorPlugConnected.stProcessedInput;

// NETWORK 14
fbOutfeedConveyorPlugConnected(
    bEnable := FALSE,
    eTypeInput := gDevice.stMachineConfig.st_I_OutfeedConveyorPlugConnected.eTypeInput,
    tTimeOnFilter := gDevice.stMachineConfig.st_I_OutfeedConveyorPlugConnected.tTimeOnFilter,
    tTimeOffFilter := gDevice.stMachineConfig.st_I_OutfeedConveyorPlugConnected.tTimeOffFilter); // FB_IO2_SingleInputCtrl
gIOFiltered.stOutfeedConveyorPlugConnected := fbOutfeedConveyorPlugConnected.stProcessedInput;

// NETWORK 15
fbAdditionalConveyorPlugConnected(
    bEnable := FALSE,
    eTypeInput := gDevice.stMachineConfig.st_I_AdditionalConveyorPlugConnected.eTypeInput,
    tTimeOnFilter := gDevice.stMachineConfig.st_I_AdditionalConveyorPlugConnected.tTimeOnFilter,
    tTimeOffFilter := gDevice.stMachineConfig.st_I_AdditionalConveyorPlugConnected.tTimeOffFilter); // FB_IO2_SingleInputCtrl
gIOFiltered.stAdditionalConveyorPlugConnected := fbAdditionalConveyorPlugConnected.stProcessedInput;
END_ACTION

ACTION CML:
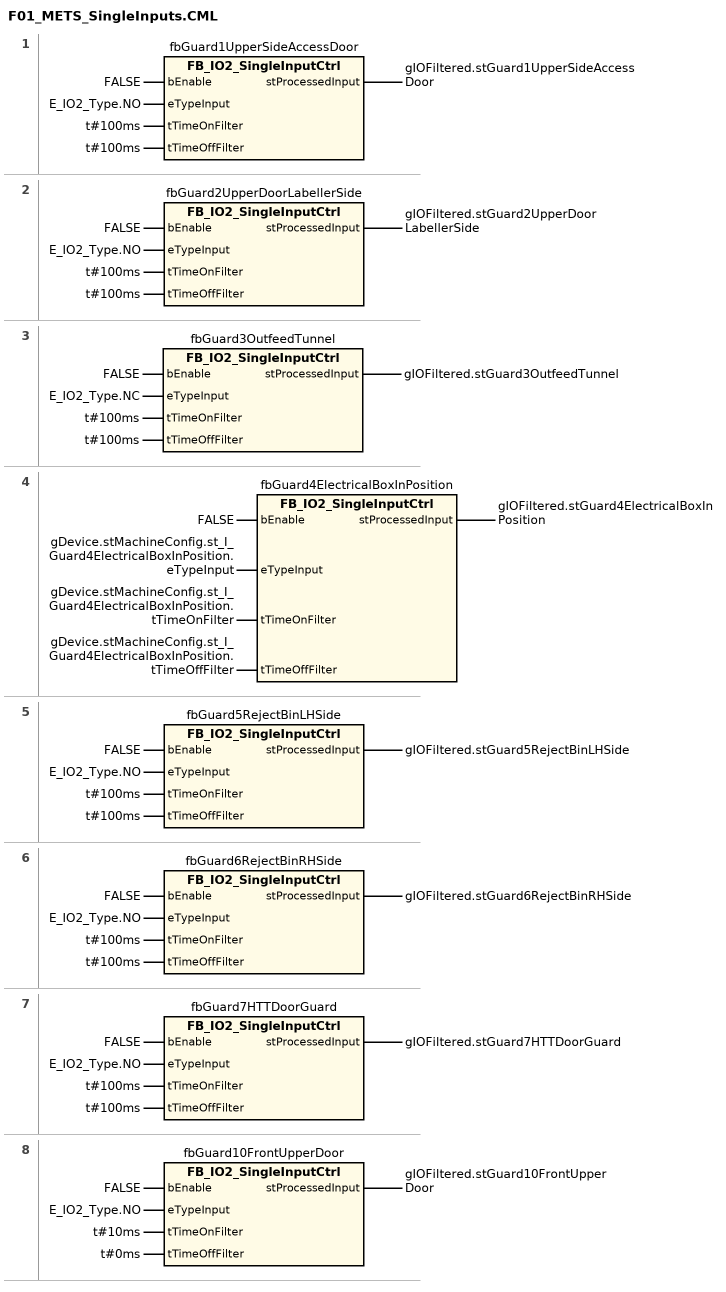
// NETWORK 1
fbGuard1UpperSideAccessDoor(
    bEnable := FALSE,
    eTypeInput := E_IO2_Type.NO,
    tTimeOnFilter := t#100ms,
    tTimeOffFilter := t#100ms); // FB_IO2_SingleInputCtrl
gIOFiltered.stGuard1UpperSideAccessDoor := fbGuard1UpperSideAccessDoor.stProcessedInput;

// NETWORK 2
fbGuard2UpperDoorLabellerSide(
    bEnable := FALSE,
    eTypeInput := E_IO2_Type.NO,
    tTimeOnFilter := t#100ms,
    tTimeOffFilter := t#100ms); // FB_IO2_SingleInputCtrl
gIOFiltered.stGuard2UpperDoorLabellerSide := fbGuard2UpperDoorLabellerSide.stProcessedInput;

// NETWORK 3
fbGuard3OutfeedTunnel(
    bEnable := FALSE,
    eTypeInput := E_IO2_Type.NC,
    tTimeOnFilter := t#100ms,
    tTimeOffFilter := t#100ms); // FB_IO2_SingleInputCtrl
gIOFiltered.stGuard3OutfeedTunnel := fbGuard3OutfeedTunnel.stProcessedInput;

// NETWORK 4
fbGuard4ElectricalBoxInPosition(
    bEnable := FALSE,
    eTypeInput := gDevice.stMachineConfig.st_I_Guard4ElectricalBoxInPosition.eTypeInput,
    tTimeOnFilter := gDevice.stMachineConfig.st_I_Guard4ElectricalBoxInPosition.tTimeOnFilter,
    tTimeOffFilter := gDevice.stMachineConfig.st_I_Guard4ElectricalBoxInPosition.tTimeOffFilter); // FB_IO2_SingleInputCtrl
gIOFiltered.stGuard4ElectricalBoxInPosition := fbGuard4ElectricalBoxInPosition.stProcessedInput;

// NETWORK 5
fbGuard5RejectBinLHSide(
    bEnable := FALSE,
    eTypeInput := E_IO2_Type.NO,
    tTimeOnFilter := t#100ms,
    tTimeOffFilter := t#100ms); // FB_IO2_SingleInputCtrl
gIOFiltered.stGuard5RejectBinLHSide := fbGuard5RejectBinLHSide.stProcessedInput;

// NETWORK 6
fbGuard6RejectBinRHSide(
    bEnable := FALSE,
    eTypeInput := E_IO2_Type.NO,
    tTimeOnFilter := t#100ms,
    tTimeOffFilter := t#100ms); // FB_IO2_SingleInputCtrl
gIOFiltered.stGuard6RejectBinRHSide := fbGuard6RejectBinRHSide.stProcessedInput;

// NETWORK 7
fbGuard7HTTDoorGuard(
    bEnable := FALSE,
    eTypeInput := E_IO2_Type.NO,
    tTimeOnFilter := t#100ms,
    tTimeOffFilter := t#100ms); // FB_IO2_SingleInputCtrl
gIOFiltered.stGuard7HTTDoorGuard := fbGuard7HTTDoorGuard.stProcessedInput;

// NETWORK 8
fbGuard10FrontUpperDoor(
    bEnable := FALSE,
    eTypeInput := E_IO2_Type.NO,
    tTimeOnFilter := t#10ms,
    tTimeOffFilter := t#0ms); // FB_IO2_SingleInputCtrl
gIOFiltered.stGuard10FrontUpperDoor := fbGuard10FrontUpperDoor.stProcessedInput;

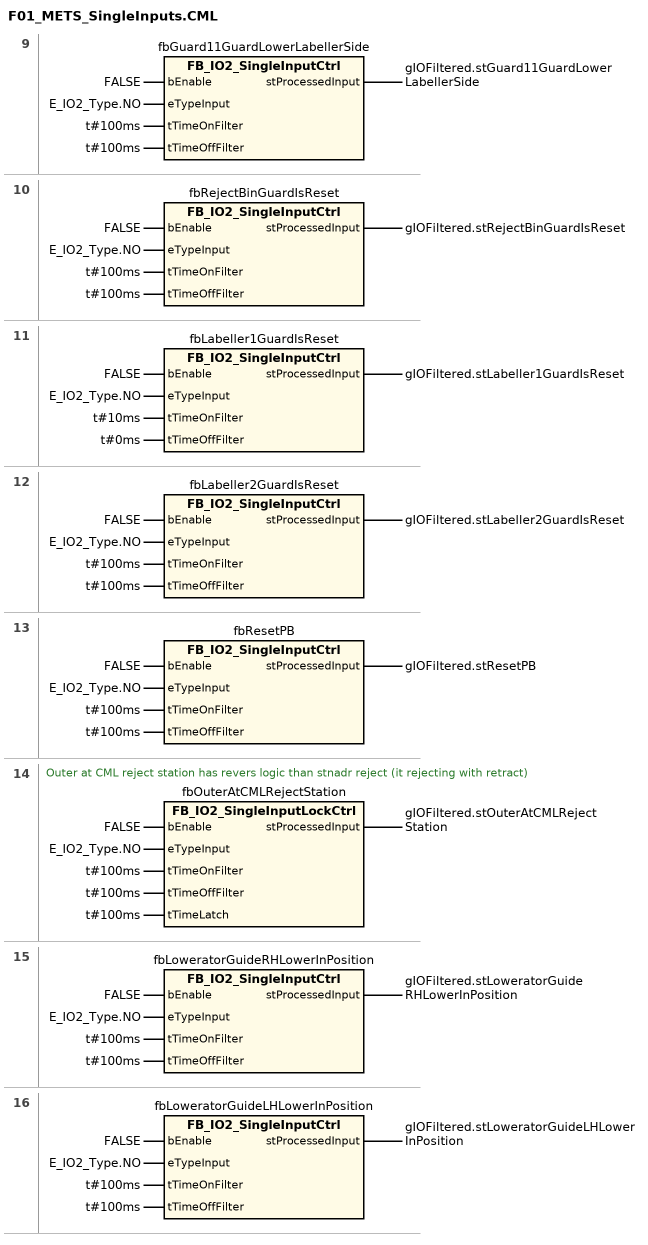
// NETWORK 9
fbGuard11GuardLowerLabellerSide(
    bEnable := FALSE,
    eTypeInput := E_IO2_Type.NO,
    tTimeOnFilter := t#100ms,
    tTimeOffFilter := t#100ms); // FB_IO2_SingleInputCtrl
gIOFiltered.stGuard11GuardLowerLabellerSide := fbGuard11GuardLowerLabellerSide.stProcessedInput;

// NETWORK 10
fbRejectBinGuardIsReset(
    bEnable := FALSE,
    eTypeInput := E_IO2_Type.NO,
    tTimeOnFilter := t#100ms,
    tTimeOffFilter := t#100ms); // FB_IO2_SingleInputCtrl
gIOFiltered.stRejectBinGuardIsReset := fbRejectBinGuardIsReset.stProcessedInput;

// NETWORK 11
fbLabeller1GuardIsReset(
    bEnable := FALSE,
    eTypeInput := E_IO2_Type.NO,
    tTimeOnFilter := t#10ms,
    tTimeOffFilter := t#0ms); // FB_IO2_SingleInputCtrl
gIOFiltered.stLabeller1GuardIsReset := fbLabeller1GuardIsReset.stProcessedInput;

// NETWORK 12
fbLabeller2GuardIsReset(
    bEnable := FALSE,
    eTypeInput := E_IO2_Type.NO,
    tTimeOnFilter := t#100ms,
    tTimeOffFilter := t#100ms); // FB_IO2_SingleInputCtrl
gIOFiltered.stLabeller2GuardIsReset := fbLabeller2GuardIsReset.stProcessedInput;

// NETWORK 13
fbResetPB(bEnable := FALSE, eTypeInput := E_IO2_Type.NO, tTimeOnFilter := t#100ms, tTimeOffFilter := t#100ms); // FB_IO2_SingleInputCtrl
gIOFiltered.stResetPB := fbResetPB.stProcessedInput;

// NETWORK 14
// Outer at CML reject station has revers logic than stnadr reject (it rejecting with retract)
fbOuterAtCMLRejectStation(
    bEnable := FALSE,
    eTypeInput := E_IO2_Type.NO,
    tTimeOnFilter := t#100ms,
    tTimeOffFilter := t#100ms,
    tTimeLatch := t#100ms); // FB_IO2_SingleInputLockCtrl
gIOFiltered.stOuterAtCMLRejectStation := fbOuterAtCMLRejectStation.stProcessedInput;

// NETWORK 15
fbLoweratorGuideRHLowerInPosition(
    bEnable := FALSE,
    eTypeInput := E_IO2_Type.NO,
    tTimeOnFilter := t#100ms,
    tTimeOffFilter := t#100ms); // FB_IO2_SingleInputCtrl
gIOFiltered.stLoweratorGuideRHLowerInPosition := fbLoweratorGuideRHLowerInPosition.stProcessedInput;

// NETWORK 16
fbLoweratorGuideLHLowerInPosition(
    bEnable := FALSE,
    eTypeInput := E_IO2_Type.NO,
    tTimeOnFilter := t#100ms,
    tTimeOffFilter := t#100ms); // FB_IO2_SingleInputCtrl
gIOFiltered.stLoweratorGuideLHLowerInPosition := fbLoweratorGuideLHLowerInPosition.stProcessedInput;
END_ACTION

ACTION CML_Drive:
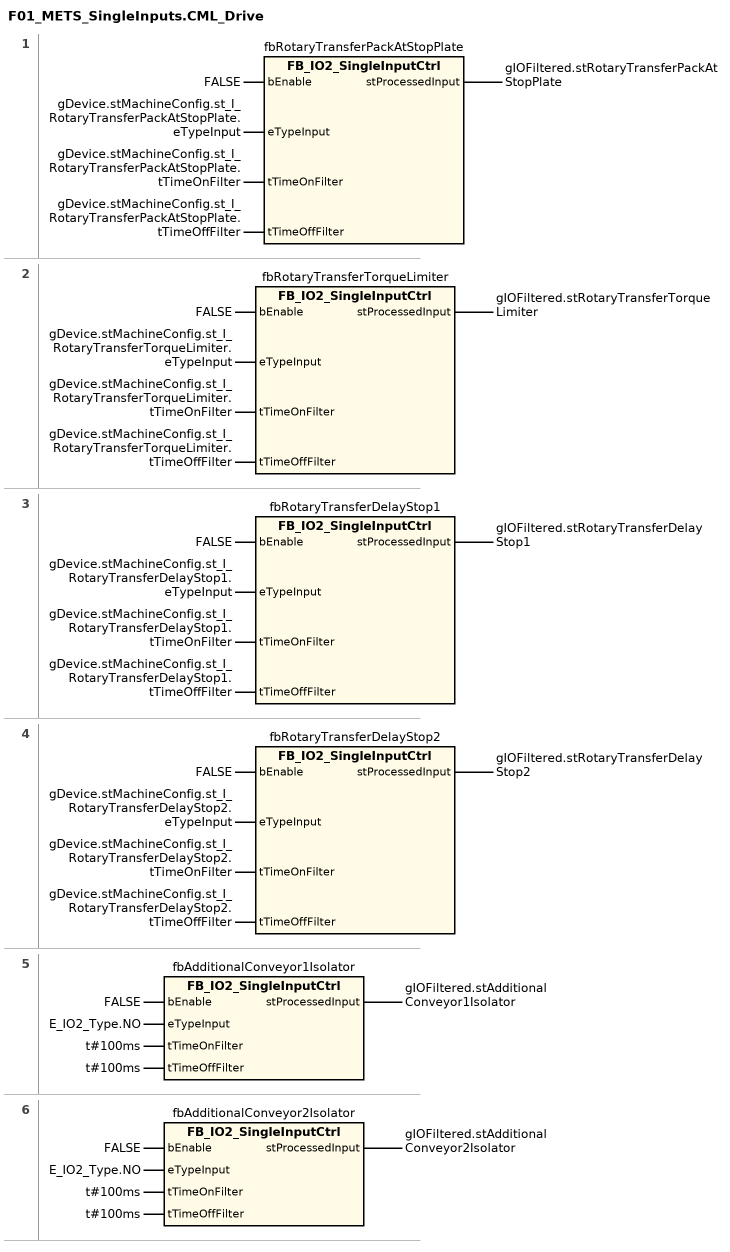
// NETWORK 1
fbRotaryTransferPackAtStopPlate(
    bEnable := FALSE,
    eTypeInput := gDevice.stMachineConfig.st_I_RotaryTransferPackAtStopPlate.eTypeInput,
    tTimeOnFilter := gDevice.stMachineConfig.st_I_RotaryTransferPackAtStopPlate.tTimeOnFilter,
    tTimeOffFilter := gDevice.stMachineConfig.st_I_RotaryTransferPackAtStopPlate.tTimeOffFilter); // FB_IO2_SingleInputCtrl
gIOFiltered.stRotaryTransferPackAtStopPlate := fbRotaryTransferPackAtStopPlate.stProcessedInput;

// NETWORK 2
fbRotaryTransferTorqueLimiter(
    bEnable := FALSE,
    eTypeInput := gDevice.stMachineConfig.st_I_RotaryTransferTorqueLimiter.eTypeInput,
    tTimeOnFilter := gDevice.stMachineConfig.st_I_RotaryTransferTorqueLimiter.tTimeOnFilter,
    tTimeOffFilter := gDevice.stMachineConfig.st_I_RotaryTransferTorqueLimiter.tTimeOffFilter); // FB_IO2_SingleInputCtrl
gIOFiltered.stRotaryTransferTorqueLimiter := fbRotaryTransferTorqueLimiter.stProcessedInput;

// NETWORK 3
fbRotaryTransferDelayStop1(
    bEnable := FALSE,
    eTypeInput := gDevice.stMachineConfig.st_I_RotaryTransferDelayStop1.eTypeInput,
    tTimeOnFilter := gDevice.stMachineConfig.st_I_RotaryTransferDelayStop1.tTimeOnFilter,
    tTimeOffFilter := gDevice.stMachineConfig.st_I_RotaryTransferDelayStop1.tTimeOffFilter); // FB_IO2_SingleInputCtrl
gIOFiltered.stRotaryTransferDelayStop1 := fbRotaryTransferDelayStop1.stProcessedInput;

// NETWORK 4
fbRotaryTransferDelayStop2(
    bEnable := FALSE,
    eTypeInput := gDevice.stMachineConfig.st_I_RotaryTransferDelayStop2.eTypeInput,
    tTimeOnFilter := gDevice.stMachineConfig.st_I_RotaryTransferDelayStop2.tTimeOnFilter,
    tTimeOffFilter := gDevice.stMachineConfig.st_I_RotaryTransferDelayStop2.tTimeOffFilter); // FB_IO2_SingleInputCtrl
gIOFiltered.stRotaryTransferDelayStop2 := fbRotaryTransferDelayStop2.stProcessedInput;

// NETWORK 5
fbAdditionalConveyor1Isolator(
    bEnable := FALSE,
    eTypeInput := E_IO2_Type.NO,
    tTimeOnFilter := t#100ms,
    tTimeOffFilter := t#100ms); // FB_IO2_SingleInputCtrl
gIOFiltered.stAdditionalConveyor1Isolator := fbAdditionalConveyor1Isolator.stProcessedInput;

// NETWORK 6
fbAdditionalConveyor2Isolator(
    bEnable := FALSE,
    eTypeInput := E_IO2_Type.NO,
    tTimeOnFilter := t#100ms,
    tTimeOffFilter := t#100ms); // FB_IO2_SingleInputCtrl
gIOFiltered.stAdditionalConveyor2Isolator := fbAdditionalConveyor2Isolator.stProcessedInput;

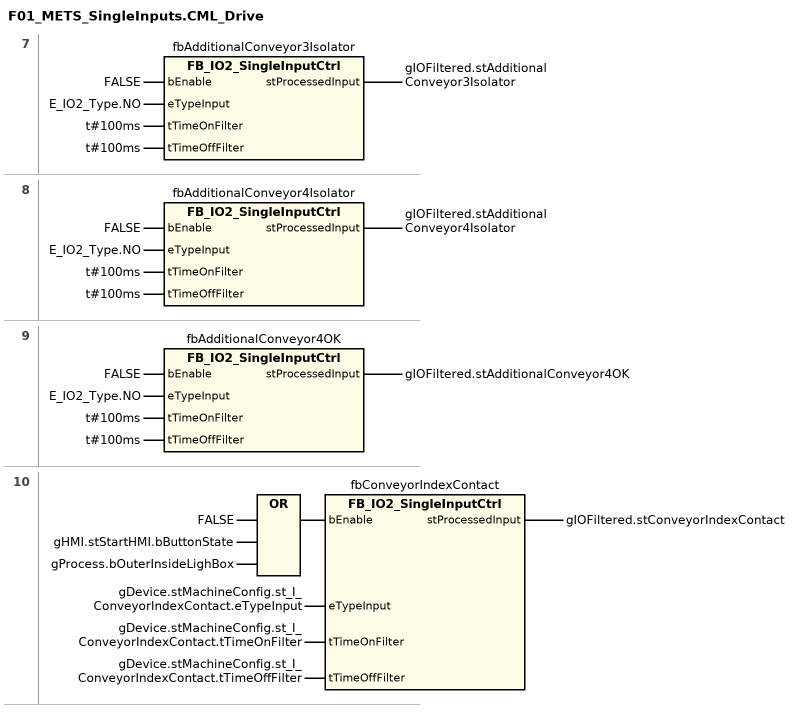
// NETWORK 7
fbAdditionalConveyor3Isolator(
    bEnable := FALSE,
    eTypeInput := E_IO2_Type.NO,
    tTimeOnFilter := t#100ms,
    tTimeOffFilter := t#100ms); // FB_IO2_SingleInputCtrl
gIOFiltered.stAdditionalConveyor3Isolator := fbAdditionalConveyor3Isolator.stProcessedInput;

// NETWORK 8
fbAdditionalConveyor4Isolator(
    bEnable := FALSE,
    eTypeInput := E_IO2_Type.NO,
    tTimeOnFilter := t#100ms,
    tTimeOffFilter := t#100ms); // FB_IO2_SingleInputCtrl
gIOFiltered.stAdditionalConveyor4Isolator := fbAdditionalConveyor4Isolator.stProcessedInput;

// NETWORK 9
fbAdditionalConveyor4OK(
    bEnable := FALSE,
    eTypeInput := E_IO2_Type.NO,
    tTimeOnFilter := t#100ms,
    tTimeOffFilter := t#100ms); // FB_IO2_SingleInputCtrl
gIOFiltered.stAdditionalConveyor4OK := fbAdditionalConveyor4OK.stProcessedInput;

// NETWORK 10
fbConveyorIndexContact(
    bEnable := FALSE OR gHMI.stStartHMI.bButtonState OR gProcess.bOuterInsideLighBox,
    eTypeInput := gDevice.stMachineConfig.st_I_ConveyorIndexContact.eTypeInput,
    tTimeOnFilter := gDevice.stMachineConfig.st_I_ConveyorIndexContact.tTimeOnFilter,
    tTimeOffFilter := gDevice.stMachineConfig.st_I_ConveyorIndexContact.tTimeOffFilter); // FB_IO2_SingleInputCtrl
gIOFiltered.stConveyorIndexContact := fbConveyorIndexContact.stProcessedInput;
END_ACTION

ACTION Cylinders:
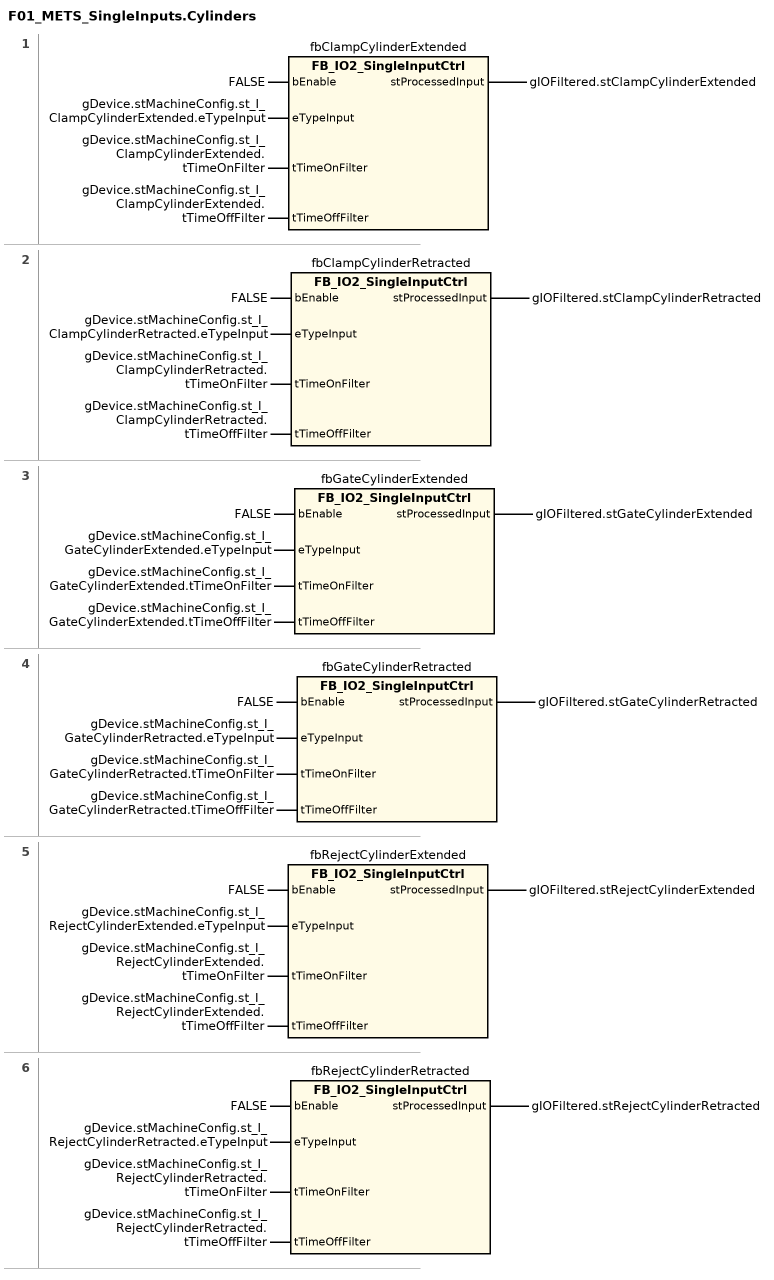
// NETWORK 1
fbClampCylinderExtended(
    bEnable := FALSE,
    eTypeInput := gDevice.stMachineConfig.st_I_ClampCylinderExtended.eTypeInput,
    tTimeOnFilter := gDevice.stMachineConfig.st_I_ClampCylinderExtended.tTimeOnFilter,
    tTimeOffFilter := gDevice.stMachineConfig.st_I_ClampCylinderExtended.tTimeOffFilter); // FB_IO2_SingleInputCtrl
gIOFiltered.stClampCylinderExtended := fbClampCylinderExtended.stProcessedInput;

// NETWORK 2
fbClampCylinderRetracted(
    bEnable := FALSE,
    eTypeInput := gDevice.stMachineConfig.st_I_ClampCylinderRetracted.eTypeInput,
    tTimeOnFilter := gDevice.stMachineConfig.st_I_ClampCylinderRetracted.tTimeOnFilter,
    tTimeOffFilter := gDevice.stMachineConfig.st_I_ClampCylinderRetracted.tTimeOffFilter); // FB_IO2_SingleInputCtrl
gIOFiltered.stClampCylinderRetracted := fbClampCylinderRetracted.stProcessedInput;

// NETWORK 3
fbGateCylinderExtended(
    bEnable := FALSE,
    eTypeInput := gDevice.stMachineConfig.st_I_GateCylinderExtended.eTypeInput,
    tTimeOnFilter := gDevice.stMachineConfig.st_I_GateCylinderExtended.tTimeOnFilter,
    tTimeOffFilter := gDevice.stMachineConfig.st_I_GateCylinderExtended.tTimeOffFilter); // FB_IO2_SingleInputCtrl
gIOFiltered.stGateCylinderExtended := fbGateCylinderExtended.stProcessedInput;

// NETWORK 4
fbGateCylinderRetracted(
    bEnable := FALSE,
    eTypeInput := gDevice.stMachineConfig.st_I_GateCylinderRetracted.eTypeInput,
    tTimeOnFilter := gDevice.stMachineConfig.st_I_GateCylinderRetracted.tTimeOnFilter,
    tTimeOffFilter := gDevice.stMachineConfig.st_I_GateCylinderRetracted.tTimeOffFilter); // FB_IO2_SingleInputCtrl
gIOFiltered.stGateCylinderRetracted := fbGateCylinderRetracted.stProcessedInput;

// NETWORK 5
fbRejectCylinderExtended(
    bEnable := FALSE,
    eTypeInput := gDevice.stMachineConfig.st_I_RejectCylinderExtended.eTypeInput,
    tTimeOnFilter := gDevice.stMachineConfig.st_I_RejectCylinderExtended.tTimeOnFilter,
    tTimeOffFilter := gDevice.stMachineConfig.st_I_RejectCylinderExtended.tTimeOffFilter); // FB_IO2_SingleInputCtrl
gIOFiltered.stRejectCylinderExtended := fbRejectCylinderExtended.stProcessedInput;

// NETWORK 6
fbRejectCylinderRetracted(
    bEnable := FALSE,
    eTypeInput := gDevice.stMachineConfig.st_I_RejectCylinderRetracted.eTypeInput,
    tTimeOnFilter := gDevice.stMachineConfig.st_I_RejectCylinderRetracted.tTimeOnFilter,
    tTimeOffFilter := gDevice.stMachineConfig.st_I_RejectCylinderRetracted.tTimeOffFilter); // FB_IO2_SingleInputCtrl
gIOFiltered.stRejectCylinderRetracted := fbRejectCylinderRetracted.stProcessedInput;

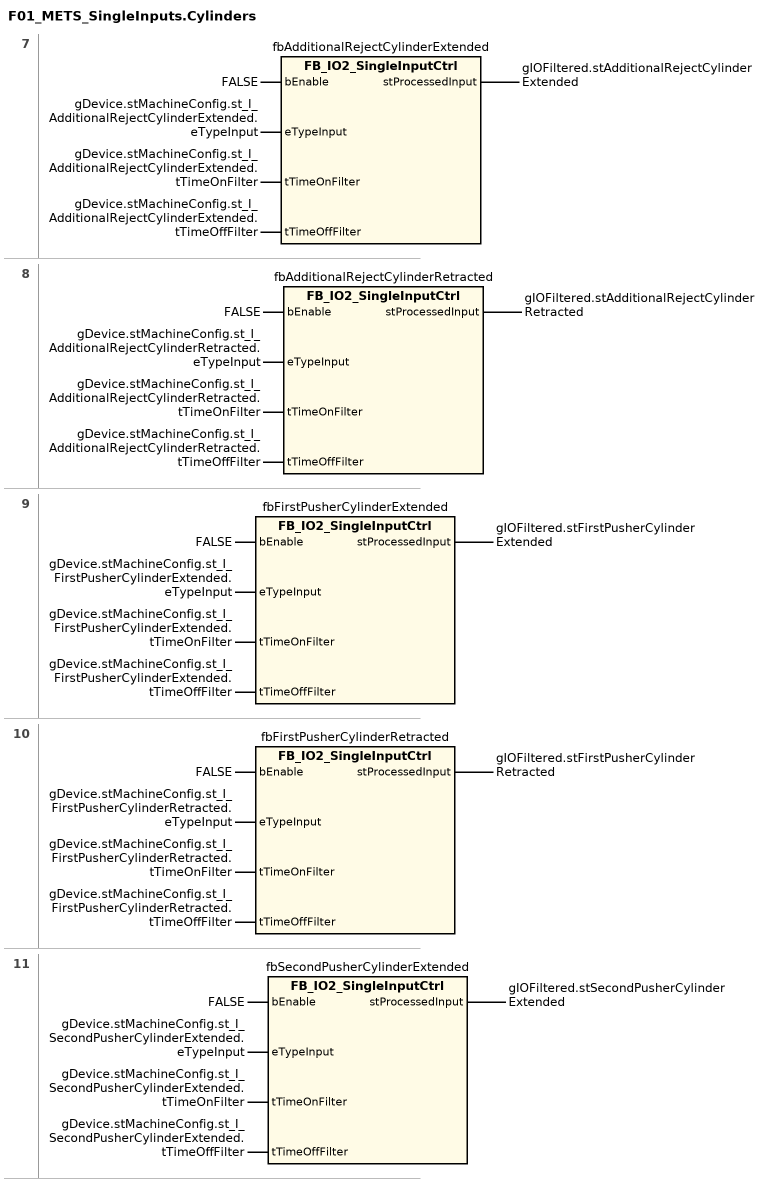
// NETWORK 7
fbAdditionalRejectCylinderExtended(
    bEnable := FALSE,
    eTypeInput := gDevice.stMachineConfig.st_I_AdditionalRejectCylinderExtended.eTypeInput,
    tTimeOnFilter := gDevice.stMachineConfig.st_I_AdditionalRejectCylinderExtended.tTimeOnFilter,
    tTimeOffFilter := gDevice.stMachineConfig.st_I_AdditionalRejectCylinderExtended.tTimeOffFilter); // FB_IO2_SingleInputCtrl
gIOFiltered.stAdditionalRejectCylinderExtended := fbAdditionalRejectCylinderExtended.stProcessedInput;

// NETWORK 8
fbAdditionalRejectCylinderRetracted(
    bEnable := FALSE,
    eTypeInput := gDevice.stMachineConfig.st_I_AdditionalRejectCylinderRetracted.eTypeInput,
    tTimeOnFilter := gDevice.stMachineConfig.st_I_AdditionalRejectCylinderRetracted.tTimeOnFilter,
    tTimeOffFilter := gDevice.stMachineConfig.st_I_AdditionalRejectCylinderRetracted.tTimeOffFilter); // FB_IO2_SingleInputCtrl
gIOFiltered.stAdditionalRejectCylinderRetracted := fbAdditionalRejectCylinderRetracted.stProcessedInput;

// NETWORK 9
fbFirstPusherCylinderExtended(
    bEnable := FALSE,
    eTypeInput := gDevice.stMachineConfig.st_I_FirstPusherCylinderExtended.eTypeInput,
    tTimeOnFilter := gDevice.stMachineConfig.st_I_FirstPusherCylinderExtended.tTimeOnFilter,
    tTimeOffFilter := gDevice.stMachineConfig.st_I_FirstPusherCylinderExtended.tTimeOffFilter); // FB_IO2_SingleInputCtrl
gIOFiltered.stFirstPusherCylinderExtended := fbFirstPusherCylinderExtended.stProcessedInput;

// NETWORK 10
fbFirstPusherCylinderRetracted(
    bEnable := FALSE,
    eTypeInput := gDevice.stMachineConfig.st_I_FirstPusherCylinderRetracted.eTypeInput,
    tTimeOnFilter := gDevice.stMachineConfig.st_I_FirstPusherCylinderRetracted.tTimeOnFilter,
    tTimeOffFilter := gDevice.stMachineConfig.st_I_FirstPusherCylinderRetracted.tTimeOffFilter); // FB_IO2_SingleInputCtrl
gIOFiltered.stFirstPusherCylinderRetracted := fbFirstPusherCylinderRetracted.stProcessedInput;

// NETWORK 11
fbSecondPusherCylinderExtended(
    bEnable := FALSE,
    eTypeInput := gDevice.stMachineConfig.st_I_SecondPusherCylinderExtended.eTypeInput,
    tTimeOnFilter := gDevice.stMachineConfig.st_I_SecondPusherCylinderExtended.tTimeOnFilter,
    tTimeOffFilter := gDevice.stMachineConfig.st_I_SecondPusherCylinderExtended.tTimeOffFilter); // FB_IO2_SingleInputCtrl
gIOFiltered.stSecondPusherCylinderExtended := fbSecondPusherCylinderExtended.stProcessedInput;

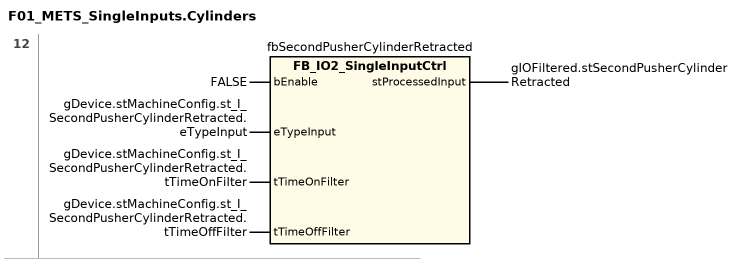
// NETWORK 12
fbSecondPusherCylinderRetracted(
    bEnable := FALSE,
    eTypeInput := gDevice.stMachineConfig.st_I_SecondPusherCylinderRetracted.eTypeInput,
    tTimeOnFilter := gDevice.stMachineConfig.st_I_SecondPusherCylinderRetracted.tTimeOnFilter,
    tTimeOffFilter := gDevice.stMachineConfig.st_I_SecondPusherCylinderRetracted.tTimeOffFilter); // FB_IO2_SingleInputCtrl
gIOFiltered.stSecondPusherCylinderRetracted := fbSecondPusherCylinderRetracted.stProcessedInput;
END_ACTION

ACTION General:
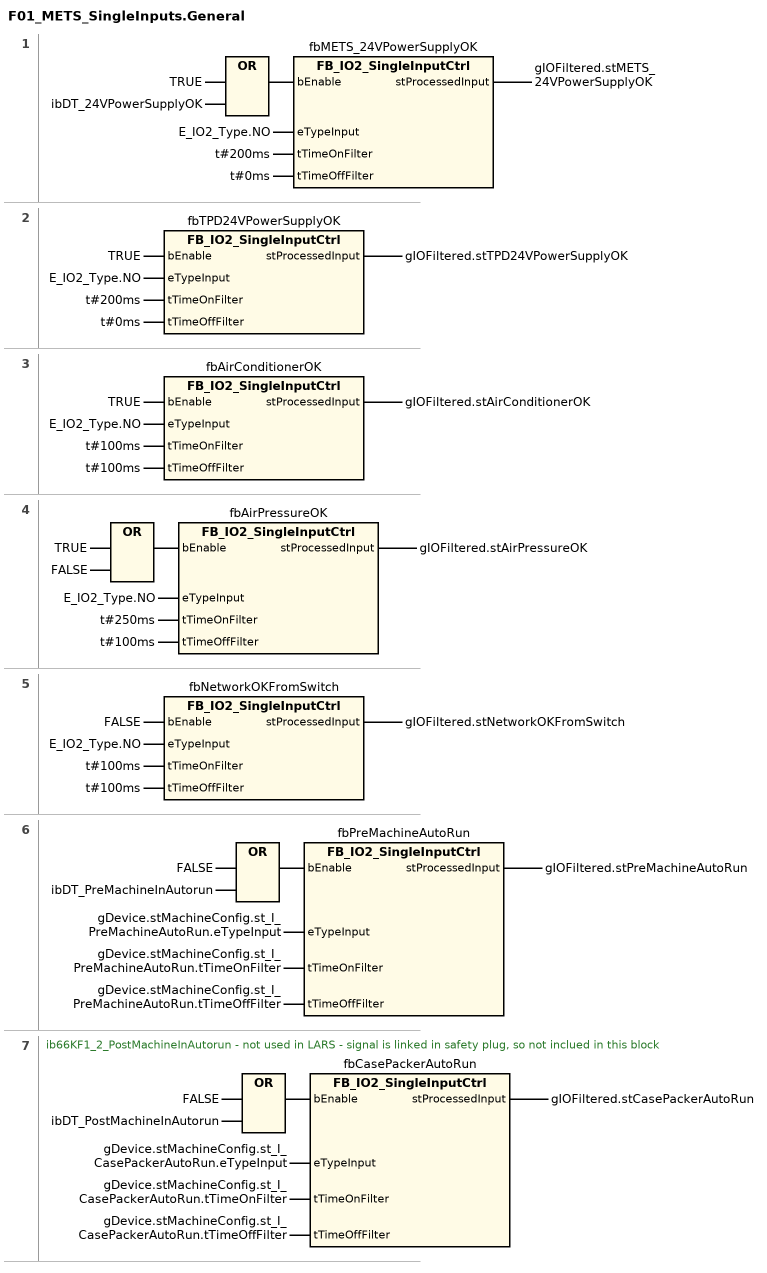
// NETWORK 1
fbMETS_24VPowerSupplyOK(
    bEnable := TRUE OR ibDT_24VPowerSupplyOK,
    eTypeInput := E_IO2_Type.NO,
    tTimeOnFilter := t#200ms,
    tTimeOffFilter := t#0ms); // FB_IO2_SingleInputCtrl
gIOFiltered.stMETS_24VPowerSupplyOK := fbMETS_24VPowerSupplyOK.stProcessedInput;

// NETWORK 2
fbTPD24VPowerSupplyOK(
    bEnable := TRUE,
    eTypeInput := E_IO2_Type.NO,
    tTimeOnFilter := t#200ms,
    tTimeOffFilter := t#0ms); // FB_IO2_SingleInputCtrl
gIOFiltered.stTPD24VPowerSupplyOK := fbTPD24VPowerSupplyOK.stProcessedInput;

// NETWORK 3
fbAirConditionerOK(
    bEnable := TRUE,
    eTypeInput := E_IO2_Type.NO,
    tTimeOnFilter := t#100ms,
    tTimeOffFilter := t#100ms); // FB_IO2_SingleInputCtrl
gIOFiltered.stAirConditionerOK := fbAirConditionerOK.stProcessedInput;

// NETWORK 4
fbAirPressureOK(
    bEnable := TRUE OR FALSE,
    eTypeInput := E_IO2_Type.NO,
    tTimeOnFilter := t#250ms,
    tTimeOffFilter := t#100ms); // FB_IO2_SingleInputCtrl
gIOFiltered.stAirPressureOK := fbAirPressureOK.stProcessedInput;

// NETWORK 5
fbNetworkOKFromSwitch(
    bEnable := FALSE,
    eTypeInput := E_IO2_Type.NO,
    tTimeOnFilter := t#100ms,
    tTimeOffFilter := t#100ms); // FB_IO2_SingleInputCtrl
gIOFiltered.stNetworkOKFromSwitch := fbNetworkOKFromSwitch.stProcessedInput;

// NETWORK 6
fbPreMachineAutoRun(
    bEnable := FALSE OR ibDT_PreMachineInAutorun,
    eTypeInput := gDevice.stMachineConfig.st_I_PreMachineAutoRun.eTypeInput,
    tTimeOnFilter := gDevice.stMachineConfig.st_I_PreMachineAutoRun.tTimeOnFilter,
    tTimeOffFilter := gDevice.stMachineConfig.st_I_PreMachineAutoRun.tTimeOffFilter); // FB_IO2_SingleInputCtrl
gIOFiltered.stPreMachineAutoRun := fbPreMachineAutoRun.stProcessedInput;

// NETWORK 7
// ib66KF1_2_PostMachineInAutorun - not used in LARS - signal is linked in safety plug, so not inclued in this block
fbCasePackerAutoRun(
    bEnable := FALSE OR ibDT_PostMachineInAutorun,
    eTypeInput := gDevice.stMachineConfig.st_I_CasePackerAutoRun.eTypeInput,
    tTimeOnFilter := gDevice.stMachineConfig.st_I_CasePackerAutoRun.tTimeOnFilter,
    tTimeOffFilter := gDevice.stMachineConfig.st_I_CasePackerAutoRun.tTimeOffFilter); // FB_IO2_SingleInputCtrl
gIOFiltered.stCasePackerAutoRun := fbCasePackerAutoRun.stProcessedInput;

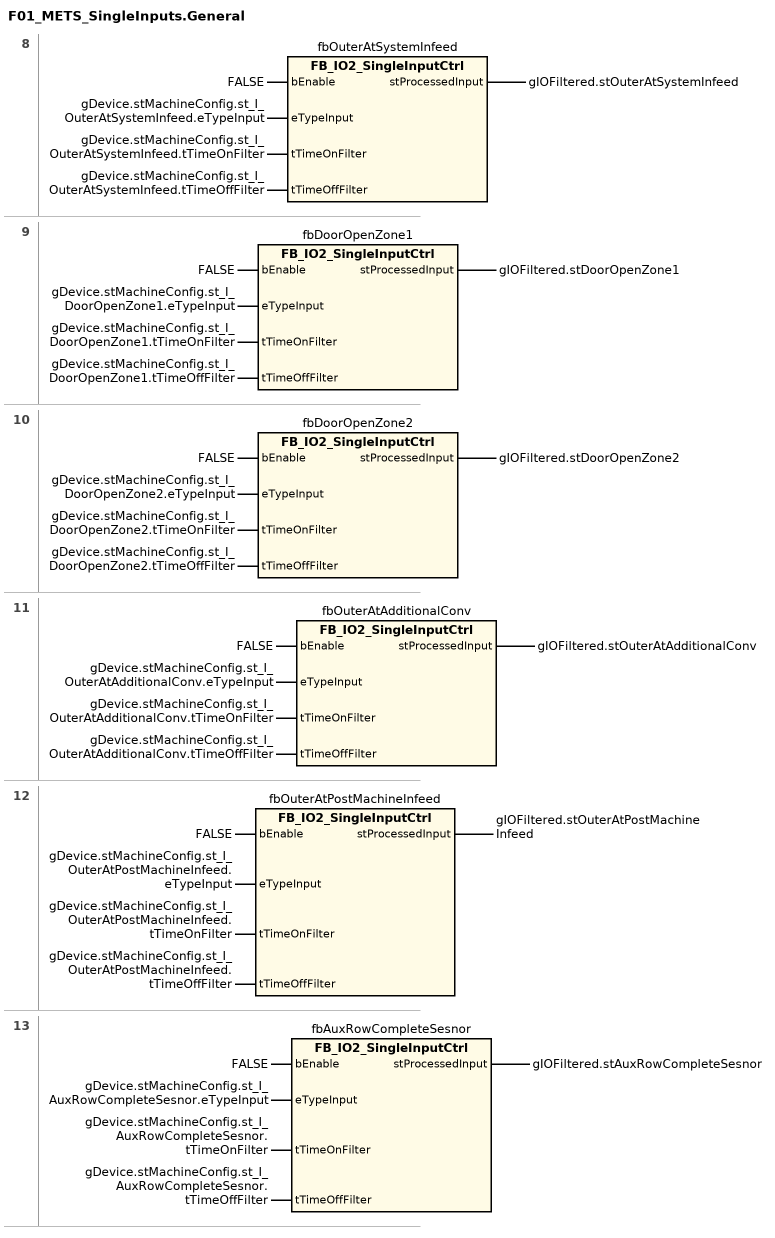
// NETWORK 8
fbOuterAtSystemInfeed(
    bEnable := FALSE,
    eTypeInput := gDevice.stMachineConfig.st_I_OuterAtSystemInfeed.eTypeInput,
    tTimeOnFilter := gDevice.stMachineConfig.st_I_OuterAtSystemInfeed.tTimeOnFilter,
    tTimeOffFilter := gDevice.stMachineConfig.st_I_OuterAtSystemInfeed.tTimeOffFilter); // FB_IO2_SingleInputCtrl
gIOFiltered.stOuterAtSystemInfeed := fbOuterAtSystemInfeed.stProcessedInput;

// NETWORK 9
fbDoorOpenZone1(
    bEnable := FALSE,
    eTypeInput := gDevice.stMachineConfig.st_I_DoorOpenZone1.eTypeInput,
    tTimeOnFilter := gDevice.stMachineConfig.st_I_DoorOpenZone1.tTimeOnFilter,
    tTimeOffFilter := gDevice.stMachineConfig.st_I_DoorOpenZone1.tTimeOffFilter); // FB_IO2_SingleInputCtrl
gIOFiltered.stDoorOpenZone1 := fbDoorOpenZone1.stProcessedInput;

// NETWORK 10
fbDoorOpenZone2(
    bEnable := FALSE,
    eTypeInput := gDevice.stMachineConfig.st_I_DoorOpenZone2.eTypeInput,
    tTimeOnFilter := gDevice.stMachineConfig.st_I_DoorOpenZone2.tTimeOnFilter,
    tTimeOffFilter := gDevice.stMachineConfig.st_I_DoorOpenZone2.tTimeOffFilter); // FB_IO2_SingleInputCtrl
gIOFiltered.stDoorOpenZone2 := fbDoorOpenZone2.stProcessedInput;

// NETWORK 11
fbOuterAtAdditionalConv(
    bEnable := FALSE,
    eTypeInput := gDevice.stMachineConfig.st_I_OuterAtAdditionalConv.eTypeInput,
    tTimeOnFilter := gDevice.stMachineConfig.st_I_OuterAtAdditionalConv.tTimeOnFilter,
    tTimeOffFilter := gDevice.stMachineConfig.st_I_OuterAtAdditionalConv.tTimeOffFilter); // FB_IO2_SingleInputCtrl
gIOFiltered.stOuterAtAdditionalConv := fbOuterAtAdditionalConv.stProcessedInput;

// NETWORK 12
fbOuterAtPostMachineInfeed(
    bEnable := FALSE,
    eTypeInput := gDevice.stMachineConfig.st_I_OuterAtPostMachineInfeed.eTypeInput,
    tTimeOnFilter := gDevice.stMachineConfig.st_I_OuterAtPostMachineInfeed.tTimeOnFilter,
    tTimeOffFilter := gDevice.stMachineConfig.st_I_OuterAtPostMachineInfeed.tTimeOffFilter); // FB_IO2_SingleInputCtrl
gIOFiltered.stOuterAtPostMachineInfeed := fbOuterAtPostMachineInfeed.stProcessedInput;

// NETWORK 13
fbAuxRowCompleteSesnor(
    bEnable := FALSE,
    eTypeInput := gDevice.stMachineConfig.st_I_AuxRowCompleteSesnor.eTypeInput,
    tTimeOnFilter := gDevice.stMachineConfig.st_I_AuxRowCompleteSesnor.tTimeOnFilter,
    tTimeOffFilter := gDevice.stMachineConfig.st_I_AuxRowCompleteSesnor.tTimeOffFilter); // FB_IO2_SingleInputCtrl
gIOFiltered.stAuxRowCompleteSesnor := fbAuxRowCompleteSesnor.stProcessedInput;

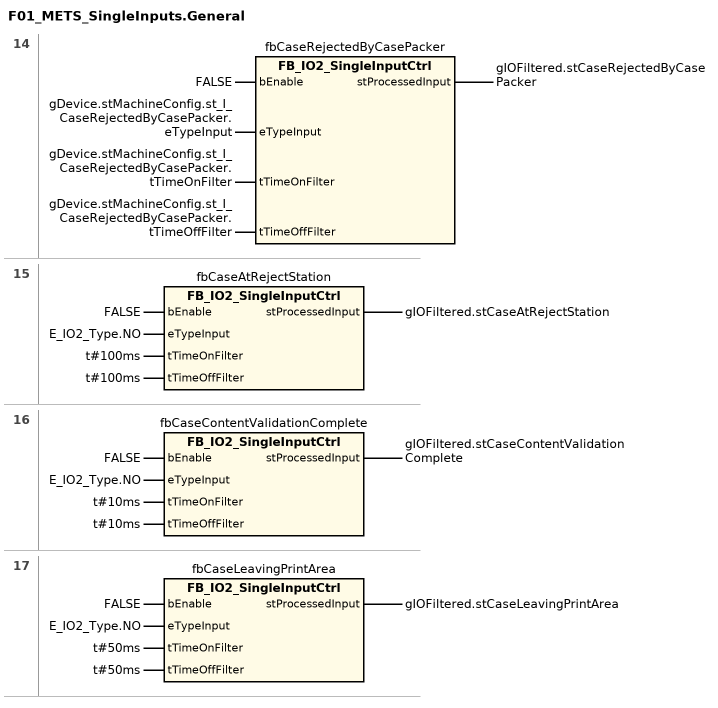
// NETWORK 14
fbCaseRejectedByCasePacker(
    bEnable := FALSE,
    eTypeInput := gDevice.stMachineConfig.st_I_CaseRejectedByCasePacker.eTypeInput,
    tTimeOnFilter := gDevice.stMachineConfig.st_I_CaseRejectedByCasePacker.tTimeOnFilter,
    tTimeOffFilter := gDevice.stMachineConfig.st_I_CaseRejectedByCasePacker.tTimeOffFilter); // FB_IO2_SingleInputCtrl
gIOFiltered.stCaseRejectedByCasePacker := fbCaseRejectedByCasePacker.stProcessedInput;

// NETWORK 15
fbCaseAtRejectStation(
    bEnable := FALSE,
    eTypeInput := E_IO2_Type.NO,
    tTimeOnFilter := t#100ms,
    tTimeOffFilter := t#100ms); // FB_IO2_SingleInputCtrl
gIOFiltered.stCaseAtRejectStation := fbCaseAtRejectStation.stProcessedInput;

// NETWORK 16
fbCaseContentValidationComplete(
    bEnable := FALSE,
    eTypeInput := E_IO2_Type.NO,
    tTimeOnFilter := t#10ms,
    tTimeOffFilter := t#10ms); // FB_IO2_SingleInputCtrl
gIOFiltered.stCaseContentValidationComplete := fbCaseContentValidationComplete.stProcessedInput;

// NETWORK 17
fbCaseLeavingPrintArea(
    bEnable := FALSE,
    eTypeInput := E_IO2_Type.NO,
    tTimeOnFilter := t#50ms,
    tTimeOffFilter := t#50ms); // FB_IO2_SingleInputCtrl
gIOFiltered.stCaseLeavingPrintArea := fbCaseLeavingPrintArea.stProcessedInput;
END_ACTION

ACTION Labellers:
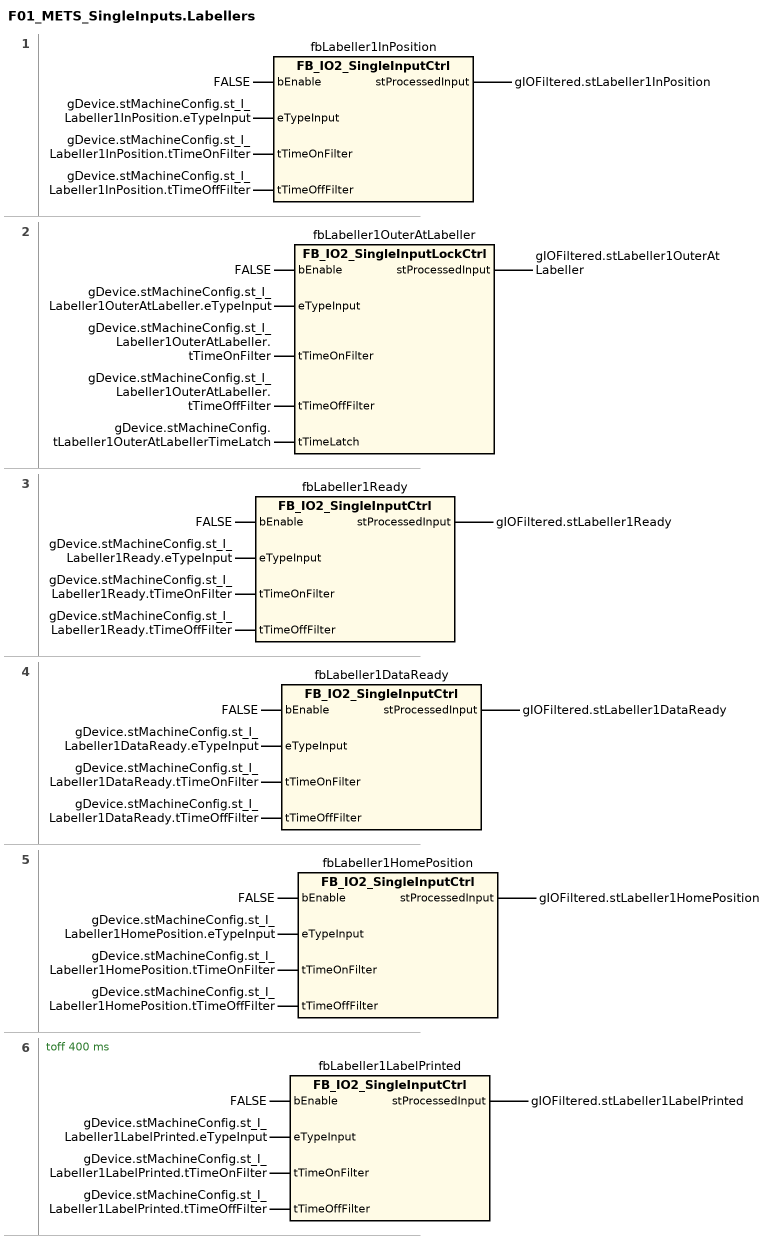
// NETWORK 1
fbLabeller1InPosition(
    bEnable := FALSE,
    eTypeInput := gDevice.stMachineConfig.st_I_Labeller1InPosition.eTypeInput,
    tTimeOnFilter := gDevice.stMachineConfig.st_I_Labeller1InPosition.tTimeOnFilter,
    tTimeOffFilter := gDevice.stMachineConfig.st_I_Labeller1InPosition.tTimeOffFilter); // FB_IO2_SingleInputCtrl
gIOFiltered.stLabeller1InPosition := fbLabeller1InPosition.stProcessedInput;

// NETWORK 2
fbLabeller1OuterAtLabeller(
    bEnable := FALSE,
    eTypeInput := gDevice.stMachineConfig.st_I_Labeller1OuterAtLabeller.eTypeInput,
    tTimeOnFilter := gDevice.stMachineConfig.st_I_Labeller1OuterAtLabeller.tTimeOnFilter,
    tTimeOffFilter := gDevice.stMachineConfig.st_I_Labeller1OuterAtLabeller.tTimeOffFilter,
    tTimeLatch := gDevice.stMachineConfig.tLabeller1OuterAtLabellerTimeLatch); // FB_IO2_SingleInputLockCtrl
gIOFiltered.stLabeller1OuterAtLabeller := fbLabeller1OuterAtLabeller.stProcessedInput;

// NETWORK 3
fbLabeller1Ready(
    bEnable := FALSE,
    eTypeInput := gDevice.stMachineConfig.st_I_Labeller1Ready.eTypeInput,
    tTimeOnFilter := gDevice.stMachineConfig.st_I_Labeller1Ready.tTimeOnFilter,
    tTimeOffFilter := gDevice.stMachineConfig.st_I_Labeller1Ready.tTimeOffFilter); // FB_IO2_SingleInputCtrl
gIOFiltered.stLabeller1Ready := fbLabeller1Ready.stProcessedInput;

// NETWORK 4
fbLabeller1DataReady(
    bEnable := FALSE,
    eTypeInput := gDevice.stMachineConfig.st_I_Labeller1DataReady.eTypeInput,
    tTimeOnFilter := gDevice.stMachineConfig.st_I_Labeller1DataReady.tTimeOnFilter,
    tTimeOffFilter := gDevice.stMachineConfig.st_I_Labeller1DataReady.tTimeOffFilter); // FB_IO2_SingleInputCtrl
gIOFiltered.stLabeller1DataReady := fbLabeller1DataReady.stProcessedInput;

// NETWORK 5
fbLabeller1HomePosition(
    bEnable := FALSE,
    eTypeInput := gDevice.stMachineConfig.st_I_Labeller1HomePosition.eTypeInput,
    tTimeOnFilter := gDevice.stMachineConfig.st_I_Labeller1HomePosition.tTimeOnFilter,
    tTimeOffFilter := gDevice.stMachineConfig.st_I_Labeller1HomePosition.tTimeOffFilter); // FB_IO2_SingleInputCtrl
gIOFiltered.stLabeller1HomePosition := fbLabeller1HomePosition.stProcessedInput;

// NETWORK 6
// toff 400 ms
fbLabeller1LabelPrinted(
    bEnable := FALSE,
    eTypeInput := gDevice.stMachineConfig.st_I_Labeller1LabelPrinted.eTypeInput,
    tTimeOnFilter := gDevice.stMachineConfig.st_I_Labeller1LabelPrinted.tTimeOnFilter,
    tTimeOffFilter := gDevice.stMachineConfig.st_I_Labeller1LabelPrinted.tTimeOffFilter); // FB_IO2_SingleInputCtrl
gIOFiltered.stLabeller1LabelPrinted := fbLabeller1LabelPrinted.stProcessedInput;

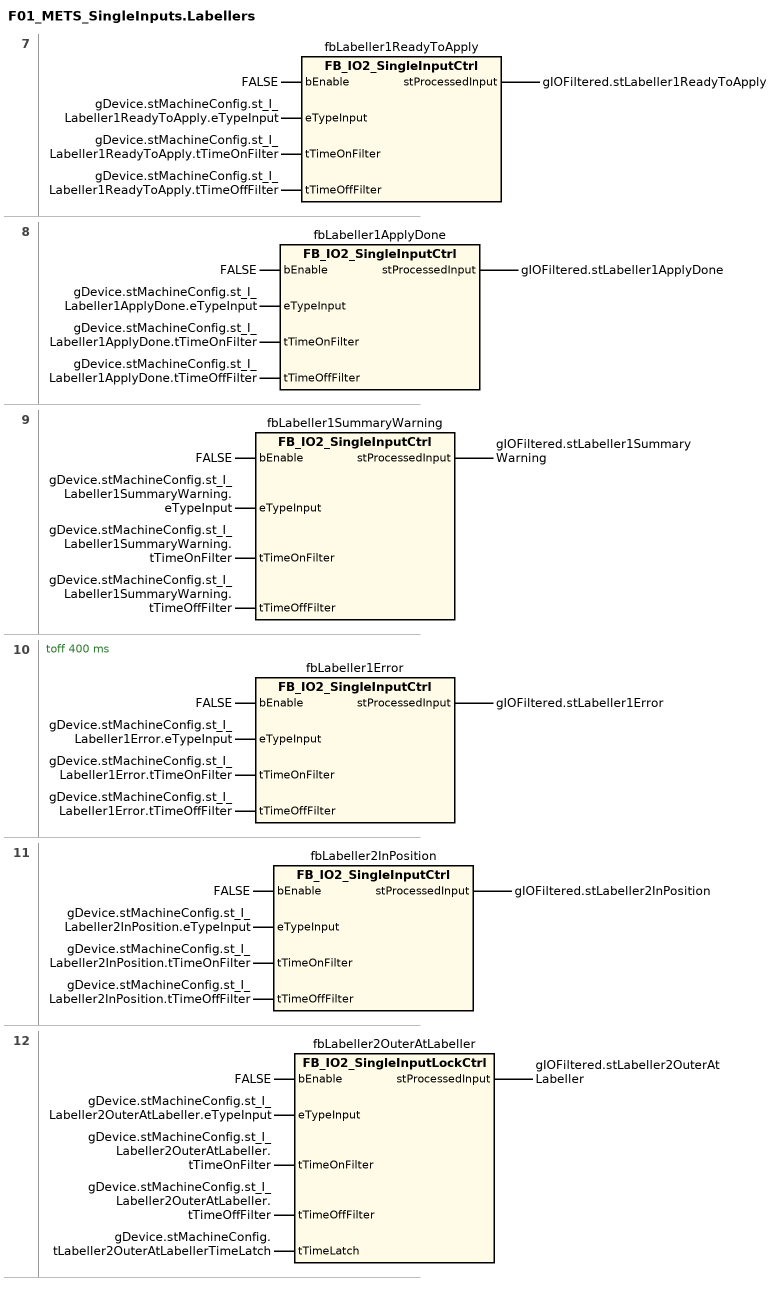
// NETWORK 7
fbLabeller1ReadyToApply(
    bEnable := FALSE,
    eTypeInput := gDevice.stMachineConfig.st_I_Labeller1ReadyToApply.eTypeInput,
    tTimeOnFilter := gDevice.stMachineConfig.st_I_Labeller1ReadyToApply.tTimeOnFilter,
    tTimeOffFilter := gDevice.stMachineConfig.st_I_Labeller1ReadyToApply.tTimeOffFilter); // FB_IO2_SingleInputCtrl
gIOFiltered.stLabeller1ReadyToApply := fbLabeller1ReadyToApply.stProcessedInput;

// NETWORK 8
fbLabeller1ApplyDone(
    bEnable := FALSE,
    eTypeInput := gDevice.stMachineConfig.st_I_Labeller1ApplyDone.eTypeInput,
    tTimeOnFilter := gDevice.stMachineConfig.st_I_Labeller1ApplyDone.tTimeOnFilter,
    tTimeOffFilter := gDevice.stMachineConfig.st_I_Labeller1ApplyDone.tTimeOffFilter); // FB_IO2_SingleInputCtrl
gIOFiltered.stLabeller1ApplyDone := fbLabeller1ApplyDone.stProcessedInput;

// NETWORK 9
fbLabeller1SummaryWarning(
    bEnable := FALSE,
    eTypeInput := gDevice.stMachineConfig.st_I_Labeller1SummaryWarning.eTypeInput,
    tTimeOnFilter := gDevice.stMachineConfig.st_I_Labeller1SummaryWarning.tTimeOnFilter,
    tTimeOffFilter := gDevice.stMachineConfig.st_I_Labeller1SummaryWarning.tTimeOffFilter); // FB_IO2_SingleInputCtrl
gIOFiltered.stLabeller1SummaryWarning := fbLabeller1SummaryWarning.stProcessedInput;

// NETWORK 10
// toff 400 ms
fbLabeller1Error(
    bEnable := FALSE,
    eTypeInput := gDevice.stMachineConfig.st_I_Labeller1Error.eTypeInput,
    tTimeOnFilter := gDevice.stMachineConfig.st_I_Labeller1Error.tTimeOnFilter,
    tTimeOffFilter := gDevice.stMachineConfig.st_I_Labeller1Error.tTimeOffFilter); // FB_IO2_SingleInputCtrl
gIOFiltered.stLabeller1Error := fbLabeller1Error.stProcessedInput;

// NETWORK 11
fbLabeller2InPosition(
    bEnable := FALSE,
    eTypeInput := gDevice.stMachineConfig.st_I_Labeller2InPosition.eTypeInput,
    tTimeOnFilter := gDevice.stMachineConfig.st_I_Labeller2InPosition.tTimeOnFilter,
    tTimeOffFilter := gDevice.stMachineConfig.st_I_Labeller2InPosition.tTimeOffFilter); // FB_IO2_SingleInputCtrl
gIOFiltered.stLabeller2InPosition := fbLabeller2InPosition.stProcessedInput;

// NETWORK 12
fbLabeller2OuterAtLabeller(
    bEnable := FALSE,
    eTypeInput := gDevice.stMachineConfig.st_I_Labeller2OuterAtLabeller.eTypeInput,
    tTimeOnFilter := gDevice.stMachineConfig.st_I_Labeller2OuterAtLabeller.tTimeOnFilter,
    tTimeOffFilter := gDevice.stMachineConfig.st_I_Labeller2OuterAtLabeller.tTimeOffFilter,
    tTimeLatch := gDevice.stMachineConfig.tLabeller2OuterAtLabellerTimeLatch); // FB_IO2_SingleInputLockCtrl
gIOFiltered.stLabeller2OuterAtLabeller := fbLabeller2OuterAtLabeller.stProcessedInput;

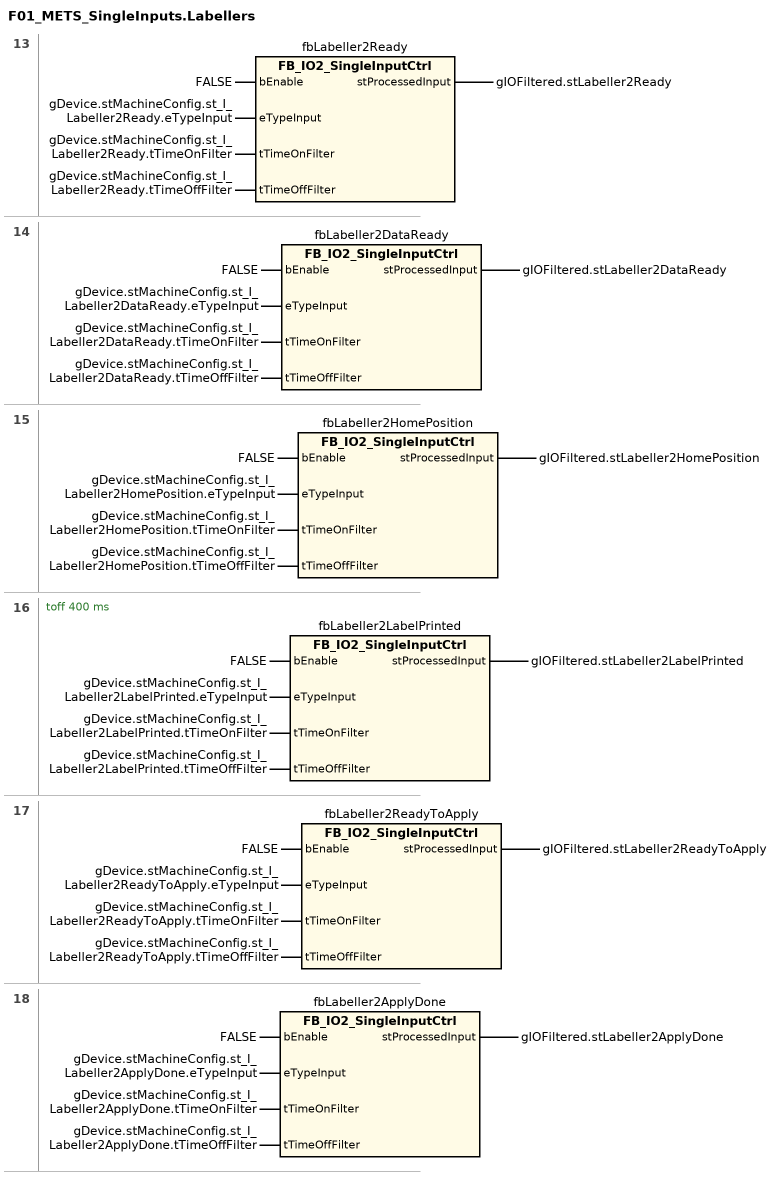
// NETWORK 13
fbLabeller2Ready(
    bEnable := FALSE,
    eTypeInput := gDevice.stMachineConfig.st_I_Labeller2Ready.eTypeInput,
    tTimeOnFilter := gDevice.stMachineConfig.st_I_Labeller2Ready.tTimeOnFilter,
    tTimeOffFilter := gDevice.stMachineConfig.st_I_Labeller2Ready.tTimeOffFilter); // FB_IO2_SingleInputCtrl
gIOFiltered.stLabeller2Ready := fbLabeller2Ready.stProcessedInput;

// NETWORK 14
fbLabeller2DataReady(
    bEnable := FALSE,
    eTypeInput := gDevice.stMachineConfig.st_I_Labeller2DataReady.eTypeInput,
    tTimeOnFilter := gDevice.stMachineConfig.st_I_Labeller2DataReady.tTimeOnFilter,
    tTimeOffFilter := gDevice.stMachineConfig.st_I_Labeller2DataReady.tTimeOffFilter); // FB_IO2_SingleInputCtrl
gIOFiltered.stLabeller2DataReady := fbLabeller2DataReady.stProcessedInput;

// NETWORK 15
fbLabeller2HomePosition(
    bEnable := FALSE,
    eTypeInput := gDevice.stMachineConfig.st_I_Labeller2HomePosition.eTypeInput,
    tTimeOnFilter := gDevice.stMachineConfig.st_I_Labeller2HomePosition.tTimeOnFilter,
    tTimeOffFilter := gDevice.stMachineConfig.st_I_Labeller2HomePosition.tTimeOffFilter); // FB_IO2_SingleInputCtrl
gIOFiltered.stLabeller2HomePosition := fbLabeller2HomePosition.stProcessedInput;

// NETWORK 16
// toff 400 ms
fbLabeller2LabelPrinted(
    bEnable := FALSE,
    eTypeInput := gDevice.stMachineConfig.st_I_Labeller2LabelPrinted.eTypeInput,
    tTimeOnFilter := gDevice.stMachineConfig.st_I_Labeller2LabelPrinted.tTimeOnFilter,
    tTimeOffFilter := gDevice.stMachineConfig.st_I_Labeller2LabelPrinted.tTimeOffFilter); // FB_IO2_SingleInputCtrl
gIOFiltered.stLabeller2LabelPrinted := fbLabeller2LabelPrinted.stProcessedInput;

// NETWORK 17
fbLabeller2ReadyToApply(
    bEnable := FALSE,
    eTypeInput := gDevice.stMachineConfig.st_I_Labeller2ReadyToApply.eTypeInput,
    tTimeOnFilter := gDevice.stMachineConfig.st_I_Labeller2ReadyToApply.tTimeOnFilter,
    tTimeOffFilter := gDevice.stMachineConfig.st_I_Labeller2ReadyToApply.tTimeOffFilter); // FB_IO2_SingleInputCtrl
gIOFiltered.stLabeller2ReadyToApply := fbLabeller2ReadyToApply.stProcessedInput;

// NETWORK 18
fbLabeller2ApplyDone(
    bEnable := FALSE,
    eTypeInput := gDevice.stMachineConfig.st_I_Labeller2ApplyDone.eTypeInput,
    tTimeOnFilter := gDevice.stMachineConfig.st_I_Labeller2ApplyDone.tTimeOnFilter,
    tTimeOffFilter := gDevice.stMachineConfig.st_I_Labeller2ApplyDone.tTimeOffFilter); // FB_IO2_SingleInputCtrl
gIOFiltered.stLabeller2ApplyDone := fbLabeller2ApplyDone.stProcessedInput;

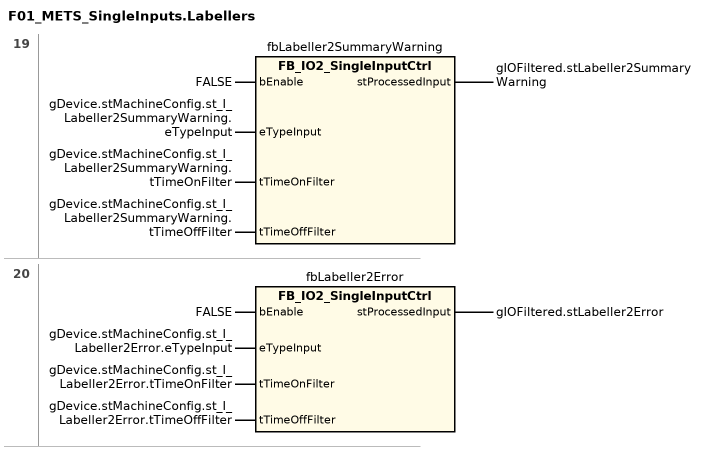
// NETWORK 19
fbLabeller2SummaryWarning(
    bEnable := FALSE,
    eTypeInput := gDevice.stMachineConfig.st_I_Labeller2SummaryWarning.eTypeInput,
    tTimeOnFilter := gDevice.stMachineConfig.st_I_Labeller2SummaryWarning.tTimeOnFilter,
    tTimeOffFilter := gDevice.stMachineConfig.st_I_Labeller2SummaryWarning.tTimeOffFilter); // FB_IO2_SingleInputCtrl
gIOFiltered.stLabeller2SummaryWarning := fbLabeller2SummaryWarning.stProcessedInput;

// NETWORK 20
fbLabeller2Error(
    bEnable := FALSE,
    eTypeInput := gDevice.stMachineConfig.st_I_Labeller2Error.eTypeInput,
    tTimeOnFilter := gDevice.stMachineConfig.st_I_Labeller2Error.tTimeOnFilter,
    tTimeOffFilter := gDevice.stMachineConfig.st_I_Labeller2Error.tTimeOffFilter); // FB_IO2_SingleInputCtrl
gIOFiltered.stLabeller2Error := fbLabeller2Error.stProcessedInput;
END_ACTION

ACTION PAOL:
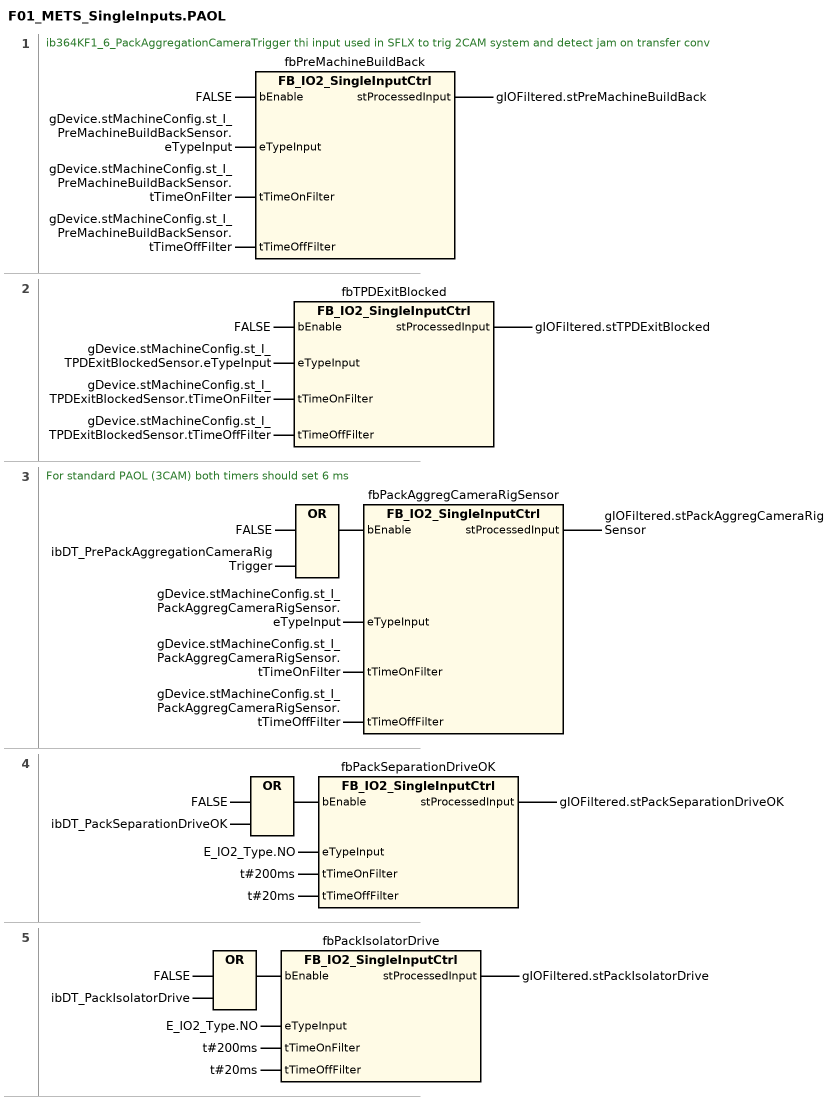
// NETWORK 1
// ib364KF1_6_PackAggregationCameraTrigger thi input used in SFLX to trig 2CAM system and detect jam on transfer conv
fbPreMachineBuildBack(
    bEnable := FALSE,
    eTypeInput := gDevice.stMachineConfig.st_I_PreMachineBuildBackSensor.eTypeInput,
    tTimeOnFilter := gDevice.stMachineConfig.st_I_PreMachineBuildBackSensor.tTimeOnFilter,
    tTimeOffFilter := gDevice.stMachineConfig.st_I_PreMachineBuildBackSensor.tTimeOffFilter); // FB_IO2_SingleInputCtrl
gIOFiltered.stPreMachineBuildBack := fbPreMachineBuildBack.stProcessedInput;

// NETWORK 2
fbTPDExitBlocked(
    bEnable := FALSE,
    eTypeInput := gDevice.stMachineConfig.st_I_TPDExitBlockedSensor.eTypeInput,
    tTimeOnFilter := gDevice.stMachineConfig.st_I_TPDExitBlockedSensor.tTimeOnFilter,
    tTimeOffFilter := gDevice.stMachineConfig.st_I_TPDExitBlockedSensor.tTimeOffFilter); // FB_IO2_SingleInputCtrl
gIOFiltered.stTPDExitBlocked := fbTPDExitBlocked.stProcessedInput;

// NETWORK 3
// For standard PAOL (3CAM) both timers should set 6 ms
fbPackAggregCameraRigSensor(
    bEnable := FALSE OR ibDT_PrePackAggregationCameraRigTrigger,
    eTypeInput := gDevice.stMachineConfig.st_I_PackAggregCameraRigSensor.eTypeInput,
    tTimeOnFilter := gDevice.stMachineConfig.st_I_PackAggregCameraRigSensor.tTimeOnFilter,
    tTimeOffFilter := gDevice.stMachineConfig.st_I_PackAggregCameraRigSensor.tTimeOffFilter); // FB_IO2_SingleInputCtrl
gIOFiltered.stPackAggregCameraRigSensor := fbPackAggregCameraRigSensor.stProcessedInput;

// NETWORK 4
fbPackSeparationDriveOK(
    bEnable := FALSE OR ibDT_PackSeparationDriveOK,
    eTypeInput := E_IO2_Type.NO,
    tTimeOnFilter := t#200ms,
    tTimeOffFilter := t#20ms); // FB_IO2_SingleInputCtrl
gIOFiltered.stPackSeparationDriveOK := fbPackSeparationDriveOK.stProcessedInput;

// NETWORK 5
fbPackIsolatorDrive(
    bEnable := FALSE OR ibDT_PackIsolatorDrive,
    eTypeInput := E_IO2_Type.NO,
    tTimeOnFilter := t#200ms,
    tTimeOffFilter := t#20ms); // FB_IO2_SingleInputCtrl
gIOFiltered.stPackIsolatorDrive := fbPackIsolatorDrive.stProcessedInput;
END_ACTION

ACTION PLAS:
